   1:  PR[GP1:91,2] = PR[GP1:90,2] + -38.074;
   1:L PR[91] 10mm/sec CNT100;
   1:  PR[GP1:91,1] = PR[GP1:90,1] + -20.726;
   1:  PR[GP1:91,2] = PR[GP1:90,2] + -40.892;
   1:L PR[91] 10mm/sec CNT100;
   1:  PR[GP1:91,1] = PR[GP1:90,1] + -15.398;
   1:  PR[GP1:91,2] = PR[GP1:90,2] + -40.986;
   1:L PR[91] 10mm/sec CNT100;
   1:  PR[GP1:91,1] = PR[GP1:90,1] + -5.344;
   1:  PR[GP1:91,2] = PR[GP1:90,2] + -40.628;
   1:L PR[91] 10mm/sec CNT100;
   1:  PR[GP1:91,1] = PR[GP1:90,1] + -1.074;
   1:  PR[GP1:91,2] = PR[GP1:90,2] + -39.306;
   1:L PR[91] 10mm/sec CNT100;
   1:  PR[GP1:91,1] = PR[GP1:90,1] + 1.895;
   1:  PR[GP1:91,2] = PR[GP1:90,2] + -39.305;
   1:L PR[91] 10mm/sec CNT100;
   1:  PR[GP1:91,1] = PR[GP1:90,1] + 6.165;
   1:  PR[GP1:91,2] = PR[GP1:90,2] + -40.627;
   1:L PR[91] 10mm/sec CNT100;
   1:  PR[GP1:91,1] = PR[GP1:90,1] + 16.219;
   1:  PR[GP1:91,2] = PR[GP1:90,2] + -40.986;
   1:L PR[91] 10mm/sec CNT100;
   1:  PR[GP1:91,1] = PR[GP1:90,1] + 21.547;
   1:  PR[GP1:91,2] = PR[GP1:90,2] + -40.892;
   1:L PR[91] 10mm/sec CNT100;
   1:  PR[GP1:91,1] = PR[GP1:90,1] + 30.135;
   1:  PR[GP1:91,2] = PR[GP1:90,2] + -38.074;
   1:L PR[91] 10mm/sec CNT100;
   1:  PR[GP1:91,1] = PR[GP1:90,1] + 35.902;
   1:  PR[GP1:91,2] = PR[GP1:90,2] + -35.950;
   1:L PR[91] 10mm/sec CNT100;
   1:  PR[GP1:91,1] = PR[GP1:90,1] + 42.200;
   1:  PR[GP1:91,2] = PR[GP1:90,2] + -30.964;
   1:L PR[91] 10mm/sec CNT100;
   1:  PR[GP1:91,1] = PR[GP1:90,1] + 47.482;
   1:  PR[GP1:91,2] = PR[GP1:90,2] + -26.602;
   1:L PR[91] 10mm/sec CNT100;
   1:  PR[GP1:91,1] = PR[GP1:90,1] + 51.199;
   1:  PR[GP1:91,2] = PR[GP1:90,2] + -20.456;
   1:L PR[91] 10mm/sec CNT100;
   1:  PR[GP1:91,1] = PR[GP1:90,1] + 54.958;
   1:  PR[GP1:91,2] = PR[GP1:90,2] + -14.112;
   1:L PR[91] 10mm/sec CNT100;
   1:  PR[GP1:91,1] = PR[GP1:90,1] + 56.363;
   1:  PR[GP1:91,2] = PR[GP1:90,2] + -6.354;
   1:L PR[91] 10mm/sec CNT100;
   1:  PR[GP1:91,1] = PR[GP1:90,1] + 57.385;
   1:  PR[GP1:91,2] = PR[GP1:90,2] + -0.011;
   1:L PR[91] 10mm/sec CNT100;
   1:  PR[GP1:91,1] = PR[GP1:90,1] + 56.882;
   1:  PR[GP1:91,2] = PR[GP1:90,2] + 2.758;
   1:L PR[91] 10mm/sec CNT100;
   1:  PR[GP1:91,1] = PR[GP1:90,1] + 56.158;
   1:  PR[GP1:91,2] = PR[GP1:90,2] + 7.602;
   1:L PR[91] 10mm/sec CNT100;
   1:  PR[GP1:91,1] = PR[GP1:90,1] + 54.959;
   1:  PR[GP1:91,2] = PR[GP1:90,2] + 14.100;
   1:L PR[91] 10mm/sec CNT100;
   1:  PR[GP1:91,1] = PR[GP1:90,1] + 51.202;
   1:  PR[GP1:91,2] = PR[GP1:90,2] + 20.445;
   1:L PR[91] 10mm/sec CNT100;
   1:  PR[GP1:91,1] = PR[GP1:90,1] + 47.484;
   1:  PR[GP1:91,2] = PR[GP1:90,2] + 26.591;
   1:L PR[91] 10mm/sec CNT100;
   1:  PR[GP1:91,1] = PR[GP1:90,1] + 42.205;
   1:  PR[GP1:91,2] = PR[GP1:90,2] + 30.953;
   1:L PR[91] 10mm/sec CNT100;
   1:  PR[GP1:91,1] = PR[GP1:90,1] + 35.906;
   1:  PR[GP1:91,2] = PR[GP1:90,2] + 35.939;
   1:L PR[91] 10mm/sec CNT100;
   1:  PR[GP1:91,1] = PR[GP1:90,1] + 30.141;
   1:  PR[GP1:91,2] = PR[GP1:90,2] + 38.065;
   1:L PR[91] 10mm/sec CNT100;
   1:  PR[GP1:91,1] = PR[GP1:90,1] + 21.552;
   1:  PR[GP1:91,2] = PR[GP1:90,2] + 40.882;
   1:L PR[91] 10mm/sec CNT100;
   1:  PR[GP1:91,1] = PR[GP1:90,1] + 16.224;
   1:  PR[GP1:91,2] = PR[GP1:90,2] + 40.978;
   1:L PR[91] 10mm/sec CNT100;
   1:  PR[GP1:91,1] = PR[GP1:90,1] + 6.166;
   1:  PR[GP1:91,2] = PR[GP1:90,2] + 40.618;
   1:L PR[91] 10mm/sec CNT100;
   1:  PR[GP1:91,1] = PR[GP1:90,1] + 1.894;
   1:  PR[GP1:91,2] = PR[GP1:90,2] + 39.305;
   1:L PR[91] 10mm/sec CNT100;
   1:  PR[GP1:91,1] = PR[GP1:90,1] + -1.017;
   1:  PR[GP1:91,2] = PR[GP1:90,2] + 39.683;
   1:  PR[GP1:91,3] = PR[GP1:90,3] + 91.770;
   1:L PR[91] 10mm/sec CNT100;
   1:  PR[GP1:91,1] = PR[GP1:90,1] + -4.695;
   1:  PR[GP1:91,2] = PR[GP1:90,2] + 40.812;
   1:L PR[91] 10mm/sec CNT100;
   1:  PR[GP1:91,1] = PR[GP1:90,1] + -15.487;
   1:  PR[GP1:91,2] = PR[GP1:90,2] + 41.199;
   1:L PR[91] 10mm/sec CNT100;
   1:  PR[GP1:91,1] = PR[GP1:90,1] + -20.161;
   1:  PR[GP1:91,2] = PR[GP1:90,2] + 41.113;
   1:L PR[91] 10mm/sec CNT100;
   1:  PR[GP1:91,1] = PR[GP1:90,1] + -29.470;
   1:  PR[GP1:91,2] = PR[GP1:90,2] + 38.060;
   1:L PR[91] 10mm/sec CNT100;
   1:  PR[GP1:91,1] = PR[GP1:90,1] + -34.602;
   1:  PR[GP1:91,2] = PR[GP1:90,2] + 36.166;
   1:L PR[91] 10mm/sec CNT100;
   1:  PR[GP1:91,1] = PR[GP1:90,1] + -41.515;
   1:  PR[GP1:91,2] = PR[GP1:90,2] + 30.696;
   1:L PR[91] 10mm/sec CNT100;
   1:  PR[GP1:91,1] = PR[GP1:90,1] + -46.261;
   1:  PR[GP1:91,2] = PR[GP1:90,2] + 26.779;
   1:L PR[91] 10mm/sec CNT100;
   1:  PR[GP1:91,1] = PR[GP1:90,1] + -50.396;
   1:  PR[GP1:91,2] = PR[GP1:90,2] + 19.939;
   1:L PR[91] 10mm/sec CNT100;
   1:  PR[GP1:91,1] = PR[GP1:90,1] + -53.792;
   1:  PR[GP1:91,2] = PR[GP1:90,2] + 14.192;
   1:L PR[91] 10mm/sec CNT100;
   1:  PR[GP1:91,1] = PR[GP1:90,1] + -55.062;
   1:  PR[GP1:91,2] = PR[GP1:90,2] + 7.190;
   1:L PR[91] 10mm/sec CNT100;
   1:  PR[GP1:91,1] = PR[GP1:90,1] + -56.220;
   1:  PR[GP1:91,2] = PR[GP1:90,2] + 0.002;
   1:L PR[91] 10mm/sec CNT100;
   1:  PR[GP1:91,1] = PR[GP1:90,1] + -55.955;
   1:  PR[GP1:91,2] = PR[GP1:90,2] + -1.459;
   1:L PR[91] 10mm/sec CNT100;
   1:  PR[GP1:91,1] = PR[GP1:90,1] + -55.141;
   1:  PR[GP1:91,2] = PR[GP1:90,2] + -6.893;
   1:L PR[91] 10mm/sec CNT100;
   1:  PR[GP1:91,1] = PR[GP1:90,1] + -53.792;
   1:  PR[GP1:91,2] = PR[GP1:90,2] + -14.202;
   1:L PR[91] 10mm/sec CNT100;
   1:  PR[GP1:91,1] = PR[GP1:90,1] + -50.394;
   1:  PR[GP1:91,2] = PR[GP1:90,2] + -19.950;
   1:L PR[91] 10mm/sec CNT100;
   1:  PR[GP1:91,1] = PR[GP1:90,1] + -46.259;
   1:  PR[GP1:91,2] = PR[GP1:90,2] + -26.790;
   1:L PR[91] 10mm/sec CNT100;
   1:  PR[GP1:91,1] = PR[GP1:90,1] + -41.511;
   1:  PR[GP1:91,2] = PR[GP1:90,2] + -30.707;
   1:L PR[91] 10mm/sec CNT100;
   1:  PR[GP1:91,1] = PR[GP1:90,1] + -34.598;
   1:  PR[GP1:91,2] = PR[GP1:90,2] + -36.177;
   1:L PR[91] 10mm/sec CNT100;
   1:  PR[GP1:91,1] = PR[GP1:90,1] + -29.465;
   1:  PR[GP1:91,2] = PR[GP1:90,2] + -38.069;
   1:L PR[91] 10mm/sec CNT100;
   1:  PR[GP1:91,1] = PR[GP1:90,1] + -20.157;
   1:  PR[GP1:91,2] = PR[GP1:90,2] + -41.123;
   1:L PR[91] 10mm/sec CNT100;
   1:  PR[GP1:91,1] = PR[GP1:90,1] + -15.482;
   1:  PR[GP1:91,2] = PR[GP1:90,2] + -41.206;
   1:L PR[91] 10mm/sec CNT100;
   1:  PR[GP1:91,1] = PR[GP1:90,1] + -4.696;
   1:  PR[GP1:91,2] = PR[GP1:90,2] + -40.821;
   1:L PR[91] 10mm/sec CNT100;
   1:  PR[GP1:91,1] = PR[GP1:90,1] + -1.019;
   1:  PR[GP1:91,2] = PR[GP1:90,2] + -39.684;
   1:L PR[91] 10mm/sec CNT100;
   1:  PR[GP1:91,1] = PR[GP1:90,1] + 1.841;
   1:L PR[91] 10mm/sec CNT100;
   1:  PR[GP1:91,1] = PR[GP1:90,1] + 5.518;
   1:  PR[GP1:91,2] = PR[GP1:90,2] + -40.821;
   1:L PR[91] 10mm/sec CNT100;
   1:  PR[GP1:91,1] = PR[GP1:90,1] + 16.304;
   1:  PR[GP1:91,2] = PR[GP1:90,2] + -41.205;
   1:L PR[91] 10mm/sec CNT100;
   1:  PR[GP1:91,1] = PR[GP1:90,1] + 20.979;
   1:  PR[GP1:91,2] = PR[GP1:90,2] + -41.123;
   1:L PR[91] 10mm/sec CNT100;
   1:  PR[GP1:91,1] = PR[GP1:90,1] + 30.286;
   1:  PR[GP1:91,2] = PR[GP1:90,2] + -38.069;
   1:L PR[91] 10mm/sec CNT100;
   1:  PR[GP1:91,1] = PR[GP1:90,1] + 35.419;
   1:  PR[GP1:91,2] = PR[GP1:90,2] + -36.178;
   1:L PR[91] 10mm/sec CNT100;
   1:  PR[GP1:91,1] = PR[GP1:90,1] + 42.331;
   1:  PR[GP1:91,2] = PR[GP1:90,2] + -30.706;
   1:L PR[91] 10mm/sec CNT100;
   1:  PR[GP1:91,1] = PR[GP1:90,1] + 47.079;
   1:  PR[GP1:91,2] = PR[GP1:90,2] + -26.786;
   1:L PR[91] 10mm/sec CNT100;
   1:  PR[GP1:91,1] = PR[GP1:90,1] + 51.215;
   1:  PR[GP1:91,2] = PR[GP1:90,2] + -19.949;
   1:L PR[91] 10mm/sec CNT100;
   1:  PR[GP1:91,1] = PR[GP1:90,1] + 54.612;
   1:  PR[GP1:91,2] = PR[GP1:90,2] + -14.214;
   1:L PR[91] 10mm/sec CNT100;
   1:  PR[GP1:91,1] = PR[GP1:90,1] + 55.883;
   1:  PR[GP1:91,2] = PR[GP1:90,2] + -7.201;
   1:L PR[91] 10mm/sec CNT100;
   1:  PR[GP1:91,1] = PR[GP1:90,1] + 57.041;
   1:  PR[GP1:91,2] = PR[GP1:90,2] + -0.011;
   1:L PR[91] 10mm/sec CNT100;
   1:  PR[GP1:91,1] = PR[GP1:90,1] + 56.775;
   1:  PR[GP1:91,2] = PR[GP1:90,2] + 1.452;
   1:L PR[91] 10mm/sec CNT100;
   1:  PR[GP1:91,1] = PR[GP1:90,1] + 55.962;
   1:  PR[GP1:91,2] = PR[GP1:90,2] + 6.892;
   1:L PR[91] 10mm/sec CNT100;
   1:  PR[GP1:91,1] = PR[GP1:90,1] + 54.614;
   1:  PR[GP1:91,2] = PR[GP1:90,2] + 14.203;
   1:L PR[91] 10mm/sec CNT100;
   1:  PR[GP1:91,1] = PR[GP1:90,1] + 51.217;
   1:  PR[GP1:91,2] = PR[GP1:90,2] + 19.938;
   1:L PR[91] 10mm/sec CNT100;
   1:  PR[GP1:91,1] = PR[GP1:90,1] + 47.081;
   1:  PR[GP1:91,2] = PR[GP1:90,2] + 26.774;
   1:L PR[91] 10mm/sec CNT100;
   1:  PR[GP1:91,1] = PR[GP1:90,1] + 42.335;
   1:  PR[GP1:91,2] = PR[GP1:90,2] + 30.696;
   1:L PR[91] 10mm/sec CNT100;
   1:  PR[GP1:91,1] = PR[GP1:90,1] + 35.423;
   1:  PR[GP1:91,2] = PR[GP1:90,2] + 36.168;
   1:L PR[91] 10mm/sec CNT100;
   1:  PR[GP1:91,1] = PR[GP1:90,1] + 30.290;
   1:  PR[GP1:91,2] = PR[GP1:90,2] + 38.060;
   1:L PR[91] 10mm/sec CNT100;
   1:  PR[GP1:91,1] = PR[GP1:90,1] + 20.982;
   1:  PR[GP1:91,2] = PR[GP1:90,2] + 41.113;
   1:L PR[91] 10mm/sec CNT100;
   1:  PR[GP1:91,1] = PR[GP1:90,1] + 16.308;
   1:  PR[GP1:91,2] = PR[GP1:90,2] + 41.198;
   1:L PR[91] 10mm/sec CNT100;
   1:  PR[GP1:91,1] = PR[GP1:90,1] + 5.517;
   1:  PR[GP1:91,2] = PR[GP1:90,2] + 40.811;
   1:L PR[91] 10mm/sec CNT100;
   1:  PR[GP1:91,1] = PR[GP1:90,1] + 1.839;
   1:  PR[GP1:91,2] = PR[GP1:90,2] + 39.683;
   1:L PR[91] 10mm/sec CNT100;
   1:  PR[GP1:91,1] = PR[GP1:90,1] + -0.962;
   1:  PR[GP1:91,2] = PR[GP1:90,2] + 40.061;
   1:  PR[GP1:91,3] = PR[GP1:90,3] + 93.100;
   1:L PR[91] 10mm/sec CNT100;
   1:  PR[GP1:91,1] = PR[GP1:90,1] + -4.046;
   1:  PR[GP1:91,2] = PR[GP1:90,2] + 41.005;
   1:L PR[91] 10mm/sec CNT100;
   1:  PR[GP1:91,1] = PR[GP1:90,1] + -15.570;
   1:  PR[GP1:91,2] = PR[GP1:90,2] + 41.418;
   1:L PR[91] 10mm/sec CNT100;
   1:  PR[GP1:91,1] = PR[GP1:90,1] + -19.591;
   1:  PR[GP1:91,2] = PR[GP1:90,2] + 41.345;
   1:L PR[91] 10mm/sec CNT100;
   1:  PR[GP1:91,1] = PR[GP1:90,1] + -29.619;
   1:  PR[GP1:91,2] = PR[GP1:90,2] + 38.056;
   1:L PR[91] 10mm/sec CNT100;
   1:  PR[GP1:91,1] = PR[GP1:90,1] + -34.119;
   1:  PR[GP1:91,2] = PR[GP1:90,2] + 36.395;
   1:L PR[91] 10mm/sec CNT100;
   1:  PR[GP1:91,1] = PR[GP1:90,1] + -41.646;
   1:  PR[GP1:91,2] = PR[GP1:90,2] + 30.439;
   1:L PR[91] 10mm/sec CNT100;
   1:  PR[GP1:91,1] = PR[GP1:90,1] + -45.858;
   1:  PR[GP1:91,2] = PR[GP1:90,2] + 26.962;
   1:L PR[91] 10mm/sec CNT100;
   1:  PR[GP1:91,1] = PR[GP1:90,1] + -50.412;
   1:  PR[GP1:91,2] = PR[GP1:90,2] + 19.431;
   1:L PR[91] 10mm/sec CNT100;
   1:  PR[GP1:91,1] = PR[GP1:90,1] + -53.447;
   1:  PR[GP1:91,2] = PR[GP1:90,2] + 14.295;
   1:L PR[91] 10mm/sec CNT100;
   1:  PR[GP1:91,1] = PR[GP1:90,1] + -54.582;
   1:  PR[GP1:91,2] = PR[GP1:90,2] + 8.036;
   1:L PR[91] 10mm/sec CNT100;
   1:  PR[GP1:91,1] = PR[GP1:90,1] + -55.878;
   1:  PR[GP1:91,2] = PR[GP1:90,2] + -0.007;
   1:L PR[91] 10mm/sec CNT100;
   1:  PR[GP1:91,1] = PR[GP1:90,1] + -54.945;
   1:  PR[GP1:91,2] = PR[GP1:90,2] + -6.182;
   1:L PR[91] 10mm/sec CNT100;
   1:  PR[GP1:91,1] = PR[GP1:90,1] + -53.447;
   1:  PR[GP1:91,2] = PR[GP1:90,2] + -14.304;
   1:L PR[91] 10mm/sec CNT100;
   1:  PR[GP1:91,1] = PR[GP1:90,1] + -50.409;
   1:  PR[GP1:91,2] = PR[GP1:90,2] + -19.442;
   1:L PR[91] 10mm/sec CNT100;
   1:  PR[GP1:91,1] = PR[GP1:90,1] + -45.856;
   1:  PR[GP1:91,2] = PR[GP1:90,2] + -26.973;
   1:L PR[91] 10mm/sec CNT100;
   1:  PR[GP1:91,1] = PR[GP1:90,1] + -41.642;
   1:  PR[GP1:91,2] = PR[GP1:90,2] + -30.450;
   1:L PR[91] 10mm/sec CNT100;
   1:  PR[GP1:91,1] = PR[GP1:90,1] + -34.116;
   1:  PR[GP1:91,2] = PR[GP1:90,2] + -36.406;
   1:L PR[91] 10mm/sec CNT100;
   1:  PR[GP1:91,1] = PR[GP1:90,1] + -29.615;
   1:  PR[GP1:91,2] = PR[GP1:90,2] + -38.065;
   1:L PR[91] 10mm/sec CNT100;
   1:  PR[GP1:91,1] = PR[GP1:90,1] + -19.588;
   1:  PR[GP1:91,2] = PR[GP1:90,2] + -41.354;
   1:L PR[91] 10mm/sec CNT100;
   1:  PR[GP1:91,1] = PR[GP1:90,1] + -15.567;
   1:  PR[GP1:91,2] = PR[GP1:90,2] + -41.425;
   1:L PR[91] 10mm/sec CNT100;
   1:  PR[GP1:91,1] = PR[GP1:90,1] + -4.049;
   1:  PR[GP1:91,2] = PR[GP1:90,2] + -41.015;
   1:L PR[91] 10mm/sec CNT100;
   1:  PR[GP1:91,1] = PR[GP1:90,1] + -0.964;
   1:  PR[GP1:91,2] = PR[GP1:90,2] + -40.063;
   1:L PR[91] 10mm/sec CNT100;
   1:  PR[GP1:91,1] = PR[GP1:90,1] + 1.786;
   1:L PR[91] 10mm/sec CNT100;
   1:  PR[GP1:91,1] = PR[GP1:90,1] + 4.871;
   1:  PR[GP1:91,2] = PR[GP1:90,2] + -41.015;
   1:L PR[91] 10mm/sec CNT100;
   1:  PR[GP1:91,1] = PR[GP1:90,1] + 16.388;
   1:  PR[GP1:91,2] = PR[GP1:90,2] + -41.425;
   1:L PR[91] 10mm/sec CNT100;
   1:  PR[GP1:91,1] = PR[GP1:90,1] + 20.410;
   1:  PR[GP1:91,2] = PR[GP1:90,2] + -41.354;
   1:L PR[91] 10mm/sec CNT100;
   1:  PR[GP1:91,1] = PR[GP1:90,1] + 30.436;
   1:  PR[GP1:91,2] = PR[GP1:90,2] + -38.065;
   1:L PR[91] 10mm/sec CNT100;
   1:  PR[GP1:91,1] = PR[GP1:90,1] + 34.937;
   1:  PR[GP1:91,2] = PR[GP1:90,2] + -36.407;
   1:L PR[91] 10mm/sec CNT100;
   1:  PR[GP1:91,1] = PR[GP1:90,1] + 42.463;
   1:  PR[GP1:91,2] = PR[GP1:90,2] + -30.449;
   1:L PR[91] 10mm/sec CNT100;
   1:  PR[GP1:91,1] = PR[GP1:90,1] + 46.677;
   1:  PR[GP1:91,2] = PR[GP1:90,2] + -26.969;
   1:L PR[91] 10mm/sec CNT100;
   1:  PR[GP1:91,1] = PR[GP1:90,1] + 51.230;
   1:  PR[GP1:91,2] = PR[GP1:90,2] + -19.442;
   1:L PR[91] 10mm/sec CNT100;
   1:  PR[GP1:91,1] = PR[GP1:90,1] + 54.267;
   1:  PR[GP1:91,2] = PR[GP1:90,2] + -14.316;
   1:L PR[91] 10mm/sec CNT100;
   1:  PR[GP1:91,1] = PR[GP1:90,1] + 55.403;
   1:  PR[GP1:91,2] = PR[GP1:90,2] + -8.047;
   1:L PR[91] 10mm/sec CNT100;
   1:  PR[GP1:91,1] = PR[GP1:90,1] + 56.699;
   1:  PR[GP1:91,2] = PR[GP1:90,2] + -0.001;
   1:L PR[91] 10mm/sec CNT100;
   1:  PR[GP1:91,1] = PR[GP1:90,1] + 55.767;
   1:  PR[GP1:91,2] = PR[GP1:90,2] + 6.180;
   1:L PR[91] 10mm/sec CNT100;
   1:  PR[GP1:91,1] = PR[GP1:90,1] + 54.268;
   1:  PR[GP1:91,2] = PR[GP1:90,2] + 14.305;
   1:L PR[91] 10mm/sec CNT100;
   1:  PR[GP1:91,1] = PR[GP1:90,1] + 51.232;
   1:  PR[GP1:91,2] = PR[GP1:90,2] + 19.431;
   1:L PR[91] 10mm/sec CNT100;
   1:  PR[GP1:91,1] = PR[GP1:90,1] + 46.679;
   1:  PR[GP1:91,2] = PR[GP1:90,2] + 26.958;
   1:L PR[91] 10mm/sec CNT100;
   1:  PR[GP1:91,1] = PR[GP1:90,1] + 42.466;
   1:  PR[GP1:91,2] = PR[GP1:90,2] + 30.439;
   1:L PR[91] 10mm/sec CNT100;
   1:  PR[GP1:91,1] = PR[GP1:90,1] + 34.940;
   1:  PR[GP1:91,2] = PR[GP1:90,2] + 36.396;
   1:L PR[91] 10mm/sec CNT100;
   1:  PR[GP1:91,1] = PR[GP1:90,1] + 30.440;
   1:  PR[GP1:91,2] = PR[GP1:90,2] + 38.056;
   1:L PR[91] 10mm/sec CNT100;
   1:  PR[GP1:91,1] = PR[GP1:90,1] + 20.413;
   1:  PR[GP1:91,2] = PR[GP1:90,2] + 41.345;
   1:L PR[91] 10mm/sec CNT100;
   1:  PR[GP1:91,1] = PR[GP1:90,1] + 16.391;
   1:  PR[GP1:91,2] = PR[GP1:90,2] + 41.418;
   1:L PR[91] 10mm/sec CNT100;
   1:  PR[GP1:91,1] = PR[GP1:90,1] + 4.868;
   1:  PR[GP1:91,2] = PR[GP1:90,2] + 41.005;
   1:L PR[91] 10mm/sec CNT100;
   1:  PR[GP1:91,1] = PR[GP1:90,1] + 1.784;
   1:  PR[GP1:91,2] = PR[GP1:90,2] + 40.061;
   1:L PR[91] 10mm/sec CNT100;
   1:  PR[GP1:91,1] = PR[GP1:90,1] + -0.907;
   1:  PR[GP1:91,2] = PR[GP1:90,2] + 40.438;
   1:  PR[GP1:91,3] = PR[GP1:90,3] + 94.430;
   1:L PR[91] 10mm/sec CNT100;
   1:  PR[GP1:91,1] = PR[GP1:90,1] + -3.397;
   1:  PR[GP1:91,2] = PR[GP1:90,2] + 41.198;
   1:L PR[91] 10mm/sec CNT100;
   1:  PR[GP1:91,1] = PR[GP1:90,1] + -15.653;
   1:  PR[GP1:91,2] = PR[GP1:90,2] + 41.638;
   1:L PR[91] 10mm/sec CNT100;
   1:  PR[GP1:91,1] = PR[GP1:90,1] + -19.021;
   1:  PR[GP1:91,2] = PR[GP1:90,2] + 41.576;
   1:L PR[91] 10mm/sec CNT100;
   1:  PR[GP1:91,1] = PR[GP1:90,1] + -29.768;
   1:  PR[GP1:91,2] = PR[GP1:90,2] + 38.052;
   1:L PR[91] 10mm/sec CNT100;
   1:  PR[GP1:91,1] = PR[GP1:90,1] + -33.636;
   1:  PR[GP1:91,2] = PR[GP1:90,2] + 36.624;
   1:L PR[91] 10mm/sec CNT100;
   1:  PR[GP1:91,1] = PR[GP1:90,1] + -41.776;
   1:  PR[GP1:91,2] = PR[GP1:90,2] + 30.183;
   1:L PR[91] 10mm/sec CNT100;
   1:  PR[GP1:91,1] = PR[GP1:90,1] + -45.455;
   1:  PR[GP1:91,2] = PR[GP1:90,2] + 27.146;
   1:L PR[91] 10mm/sec CNT100;
   1:  PR[GP1:91,1] = PR[GP1:90,1] + -50.427;
   1:  PR[GP1:91,2] = PR[GP1:90,2] + 18.924;
   1:L PR[91] 10mm/sec CNT100;
   1:  PR[GP1:91,1] = PR[GP1:90,1] + -53.101;
   1:  PR[GP1:91,2] = PR[GP1:90,2] + 14.398;
   1:L PR[91] 10mm/sec CNT100;
   1:  PR[GP1:91,1] = PR[GP1:90,1] + -54.101;
   1:  PR[GP1:91,2] = PR[GP1:90,2] + 8.883;
   1:L PR[91] 10mm/sec CNT100;
   1:  PR[GP1:91,1] = PR[GP1:90,1] + -55.310;
   1:  PR[GP1:91,2] = PR[GP1:90,2] + 1.381;
   1:L PR[91] 10mm/sec CNT100;
   1:  PR[GP1:91,1] = PR[GP1:90,1] + -55.567;
   1:  PR[GP1:91,2] = PR[GP1:90,2] + -0.015;
   1:L PR[91] 10mm/sec CNT100;
   1:  PR[GP1:91,1] = PR[GP1:90,1] + -54.750;
   1:  PR[GP1:91,2] = PR[GP1:90,2] + -5.473;
   1:L PR[91] 10mm/sec CNT100;
   1:  PR[GP1:91,1] = PR[GP1:90,1] + -53.101;
   1:  PR[GP1:91,2] = PR[GP1:90,2] + -14.407;
   1:L PR[91] 10mm/sec CNT100;
   1:  PR[GP1:91,1] = PR[GP1:90,1] + -50.425;
   1:  PR[GP1:91,2] = PR[GP1:90,2] + -18.935;
   1:L PR[91] 10mm/sec CNT100;
   1:  PR[GP1:91,1] = PR[GP1:90,1] + -45.454;
   1:  PR[GP1:91,2] = PR[GP1:90,2] + -27.156;
   1:L PR[91] 10mm/sec CNT100;
   1:  PR[GP1:91,1] = PR[GP1:90,1] + -41.773;
   1:  PR[GP1:91,2] = PR[GP1:90,2] + -30.193;
   1:L PR[91] 10mm/sec CNT100;
   1:  PR[GP1:91,1] = PR[GP1:90,1] + -33.634;
   1:  PR[GP1:91,2] = PR[GP1:90,2] + -36.634;
   1:L PR[91] 10mm/sec CNT100;
   1:  PR[GP1:91,1] = PR[GP1:90,1] + -29.765;
   1:  PR[GP1:91,2] = PR[GP1:90,2] + -38.060;
   1:L PR[91] 10mm/sec CNT100;
   1:  PR[GP1:91,1] = PR[GP1:90,1] + -19.020;
   1:  PR[GP1:91,2] = PR[GP1:90,2] + -41.585;
   1:L PR[91] 10mm/sec CNT100;
   1:  PR[GP1:91,1] = PR[GP1:90,1] + -15.651;
   1:  PR[GP1:91,2] = PR[GP1:90,2] + -41.645;
   1:L PR[91] 10mm/sec CNT100;
   1:  PR[GP1:91,1] = PR[GP1:90,1] + -3.401;
   1:  PR[GP1:91,2] = PR[GP1:90,2] + -41.208;
   1:L PR[91] 10mm/sec CNT100;
   1:  PR[GP1:91,1] = PR[GP1:90,1] + -0.908;
   1:  PR[GP1:91,2] = PR[GP1:90,2] + -40.442;
   1:L PR[91] 10mm/sec CNT100;
   1:  PR[GP1:91,1] = PR[GP1:90,1] + 1.731;
   1:  PR[GP1:91,2] = PR[GP1:90,2] + -40.441;
   1:L PR[91] 10mm/sec CNT100;
   1:  PR[GP1:91,1] = PR[GP1:90,1] + 4.224;
   1:  PR[GP1:91,2] = PR[GP1:90,2] + -41.208;
   1:L PR[91] 10mm/sec CNT100;
   1:  PR[GP1:91,1] = PR[GP1:90,1] + 16.473;
   1:  PR[GP1:91,2] = PR[GP1:90,2] + -41.645;
   1:L PR[91] 10mm/sec CNT100;
   1:  PR[GP1:91,1] = PR[GP1:90,1] + 19.842;
   1:  PR[GP1:91,2] = PR[GP1:90,2] + -41.585;
   1:L PR[91] 10mm/sec CNT100;
   1:  PR[GP1:91,1] = PR[GP1:90,1] + 30.586;
   1:  PR[GP1:91,2] = PR[GP1:90,2] + -38.060;
   1:L PR[91] 10mm/sec CNT100;
   1:  PR[GP1:91,1] = PR[GP1:90,1] + 34.455;
   1:  PR[GP1:91,2] = PR[GP1:90,2] + -36.635;
   1:L PR[91] 10mm/sec CNT100;
   1:  PR[GP1:91,1] = PR[GP1:90,1] + 42.594;
   1:  PR[GP1:91,2] = PR[GP1:90,2] + -30.192;
   1:L PR[91] 10mm/sec CNT100;
   1:  PR[GP1:91,1] = PR[GP1:90,1] + 46.275;
   1:  PR[GP1:91,2] = PR[GP1:90,2] + -27.152;
   1:L PR[91] 10mm/sec CNT100;
   1:  PR[GP1:91,1] = PR[GP1:90,1] + 51.246;
   1:  PR[GP1:91,2] = PR[GP1:90,2] + -18.934;
   1:L PR[91] 10mm/sec CNT100;
   1:  PR[GP1:91,1] = PR[GP1:90,1] + 53.922;
   1:  PR[GP1:91,2] = PR[GP1:90,2] + -14.418;
   1:L PR[91] 10mm/sec CNT100;
   1:  PR[GP1:91,1] = PR[GP1:90,1] + 54.922;
   1:  PR[GP1:91,2] = PR[GP1:90,2] + -8.894;
   1:L PR[91] 10mm/sec CNT100;
   1:  PR[GP1:91,1] = PR[GP1:90,1] + 56.131;
   1:  PR[GP1:91,2] = PR[GP1:90,2] + -1.390;
   1:L PR[91] 10mm/sec CNT100;
   1:  PR[GP1:91,1] = PR[GP1:90,1] + 56.388;
   1:  PR[GP1:91,2] = PR[GP1:90,2] + 0.006;
   1:L PR[91] 10mm/sec CNT100;
   1:  PR[GP1:91,1] = PR[GP1:90,1] + 55.571;
   1:  PR[GP1:91,2] = PR[GP1:90,2] + 5.470;
   1:L PR[91] 10mm/sec CNT100;
   1:  PR[GP1:91,1] = PR[GP1:90,1] + 53.922;
   1:  PR[GP1:91,2] = PR[GP1:90,2] + 14.407;
   1:L PR[91] 10mm/sec CNT100;
   1:  PR[GP1:91,1] = PR[GP1:90,1] + 51.248;
   1:  PR[GP1:91,2] = PR[GP1:90,2] + 18.924;
   1:L PR[91] 10mm/sec CNT100;
   1:  PR[GP1:91,1] = PR[GP1:90,1] + 46.276;
   1:  PR[GP1:91,2] = PR[GP1:90,2] + 27.142;
   1:L PR[91] 10mm/sec CNT100;
   1:  PR[GP1:91,1] = PR[GP1:90,1] + 42.596;
   1:  PR[GP1:91,2] = PR[GP1:90,2] + 30.182;
   1:L PR[91] 10mm/sec CNT100;
   1:  PR[GP1:91,1] = PR[GP1:90,1] + 34.457;
   1:  PR[GP1:91,2] = PR[GP1:90,2] + 36.625;
   1:L PR[91] 10mm/sec CNT100;
   1:  PR[GP1:91,1] = PR[GP1:90,1] + 30.589;
   1:  PR[GP1:91,2] = PR[GP1:90,2] + 38.051;
   1:L PR[91] 10mm/sec CNT100;
   1:  PR[GP1:91,1] = PR[GP1:90,1] + 19.843;
   1:  PR[GP1:91,2] = PR[GP1:90,2] + 41.576;
   1:L PR[91] 10mm/sec CNT100;
   1:  PR[GP1:91,1] = PR[GP1:90,1] + 16.475;
   1:  PR[GP1:91,2] = PR[GP1:90,2] + 41.637;
   1:L PR[91] 10mm/sec CNT100;
   1:  PR[GP1:91,1] = PR[GP1:90,1] + 4.220;
   1:  PR[GP1:91,2] = PR[GP1:90,2] + 41.198;
   1:L PR[91] 10mm/sec CNT100;
   1:  PR[GP1:91,1] = PR[GP1:90,1] + 1.729;
   1:  PR[GP1:91,2] = PR[GP1:90,2] + 40.438;
   1:L PR[91] 10mm/sec CNT100;
   1:  PR[GP1:91,1] = PR[GP1:90,1] + -0.851;
   1:  PR[GP1:91,2] = PR[GP1:90,2] + 40.816;
   1:  PR[GP1:91,3] = PR[GP1:90,3] + 95.760;
   1:L PR[91] 10mm/sec CNT100;
   1:  PR[GP1:91,1] = PR[GP1:90,1] + -2.748;
   1:  PR[GP1:91,2] = PR[GP1:90,2] + 41.391;
   1:L PR[91] 10mm/sec CNT100;
   1:  PR[GP1:91,1] = PR[GP1:90,1] + -15.736;
   1:  PR[GP1:91,2] = PR[GP1:90,2] + 41.857;
   1:L PR[91] 10mm/sec CNT100;
   1:  PR[GP1:91,1] = PR[GP1:90,1] + -18.451;
   1:  PR[GP1:91,2] = PR[GP1:90,2] + 41.807;
   1:L PR[91] 10mm/sec CNT100;
   1:  PR[GP1:91,1] = PR[GP1:90,1] + -29.917;
   1:  PR[GP1:91,2] = PR[GP1:90,2] + 38.047;
   1:L PR[91] 10mm/sec CNT100;
   1:  PR[GP1:91,1] = PR[GP1:90,1] + -33.153;
   1:  PR[GP1:91,2] = PR[GP1:90,2] + 36.853;
   1:L PR[91] 10mm/sec CNT100;
   1:  PR[GP1:91,1] = PR[GP1:90,1] + -41.907;
   1:  PR[GP1:91,2] = PR[GP1:90,2] + 29.926;
   1:L PR[91] 10mm/sec CNT100;
   1:  PR[GP1:91,1] = PR[GP1:90,1] + -45.053;
   1:  PR[GP1:91,2] = PR[GP1:90,2] + 27.329;
   1:L PR[91] 10mm/sec CNT100;
   1:  PR[GP1:91,1] = PR[GP1:90,1] + -50.442;
   1:  PR[GP1:91,2] = PR[GP1:90,2] + 18.416;
   1:L PR[91] 10mm/sec CNT100;
   1:  PR[GP1:91,1] = PR[GP1:90,1] + -52.756;
   1:  PR[GP1:91,2] = PR[GP1:90,2] + 14.501;
   1:L PR[91] 10mm/sec CNT100;
   1:  PR[GP1:91,1] = PR[GP1:90,1] + -53.621;
   1:  PR[GP1:91,2] = PR[GP1:90,2] + 9.729;
   1:L PR[91] 10mm/sec CNT100;
   1:  PR[GP1:91,1] = PR[GP1:90,1] + -54.670;
   1:  PR[GP1:91,2] = PR[GP1:90,2] + 3.218;
   1:L PR[91] 10mm/sec CNT100;
   1:  PR[GP1:91,1] = PR[GP1:90,1] + -55.265;
   1:  PR[GP1:91,2] = PR[GP1:90,2] + -0.015;
   1:L PR[91] 10mm/sec CNT100;
   1:  PR[GP1:91,1] = PR[GP1:90,1] + -54.554;
   1:  PR[GP1:91,2] = PR[GP1:90,2] + -4.763;
   1:L PR[91] 10mm/sec CNT100;
   1:  PR[GP1:91,1] = PR[GP1:90,1] + -52.756;
   1:  PR[GP1:91,2] = PR[GP1:90,2] + -14.510;
   1:L PR[91] 10mm/sec CNT100;
   1:  PR[GP1:91,1] = PR[GP1:90,1] + -50.440;
   1:  PR[GP1:91,2] = PR[GP1:90,2] + -18.427;
   1:L PR[91] 10mm/sec CNT100;
   1:  PR[GP1:91,1] = PR[GP1:90,1] + -45.052;
   1:  PR[GP1:91,2] = PR[GP1:90,2] + -27.339;
   1:L PR[91] 10mm/sec CNT100;
   1:  PR[GP1:91,1] = PR[GP1:90,1] + -41.904;
   1:  PR[GP1:91,2] = PR[GP1:90,2] + -29.936;
   1:L PR[91] 10mm/sec CNT100;
   1:  PR[GP1:91,1] = PR[GP1:90,1] + -33.151;
   1:  PR[GP1:91,2] = PR[GP1:90,2] + -36.863;
   1:L PR[91] 10mm/sec CNT100;
   1:  PR[GP1:91,1] = PR[GP1:90,1] + -29.915;
   1:  PR[GP1:91,2] = PR[GP1:90,2] + -38.056;
   1:L PR[91] 10mm/sec CNT100;
   1:  PR[GP1:91,1] = PR[GP1:90,1] + -18.451;
   1:  PR[GP1:91,2] = PR[GP1:90,2] + -41.817;
   1:L PR[91] 10mm/sec CNT100;
   1:  PR[GP1:91,1] = PR[GP1:90,1] + -15.736;
   1:  PR[GP1:91,2] = PR[GP1:90,2] + -41.865;
   1:L PR[91] 10mm/sec CNT100;
   1:  PR[GP1:91,1] = PR[GP1:90,1] + -2.753;
   1:  PR[GP1:91,2] = PR[GP1:90,2] + -41.402;
   1:L PR[91] 10mm/sec CNT100;
   1:  PR[GP1:91,1] = PR[GP1:90,1] + -0.853;
   1:  PR[GP1:91,2] = PR[GP1:90,2] + -40.820;
   1:L PR[91] 10mm/sec CNT100;
   1:  PR[GP1:91,1] = PR[GP1:90,1] + 1.676;
   1:L PR[91] 10mm/sec CNT100;
   1:  PR[GP1:91,1] = PR[GP1:90,1] + 3.576;
   1:  PR[GP1:91,2] = PR[GP1:90,2] + -41.402;
   1:L PR[91] 10mm/sec CNT100;
   1:  PR[GP1:91,1] = PR[GP1:90,1] + 16.558;
   1:  PR[GP1:91,2] = PR[GP1:90,2] + -41.864;
   1:L PR[91] 10mm/sec CNT100;
   1:  PR[GP1:91,1] = PR[GP1:90,1] + 19.273;
   1:  PR[GP1:91,2] = PR[GP1:90,2] + -41.817;
   1:L PR[91] 10mm/sec CNT100;
   1:  PR[GP1:91,1] = PR[GP1:90,1] + 30.737;
   1:  PR[GP1:91,2] = PR[GP1:90,2] + -38.056;
   1:L PR[91] 10mm/sec CNT100;
   1:  PR[GP1:91,1] = PR[GP1:90,1] + 33.973;
   1:  PR[GP1:91,2] = PR[GP1:90,2] + -36.863;
   1:L PR[91] 10mm/sec CNT100;
   1:  PR[GP1:91,1] = PR[GP1:90,1] + 42.725;
   1:  PR[GP1:91,2] = PR[GP1:90,2] + -29.935;
   1:L PR[91] 10mm/sec CNT100;
   1:  PR[GP1:91,1] = PR[GP1:90,1] + 45.873;
   1:  PR[GP1:91,2] = PR[GP1:90,2] + -27.335;
   1:L PR[91] 10mm/sec CNT100;
   1:  PR[GP1:91,1] = PR[GP1:90,1] + 51.261;
   1:  PR[GP1:91,2] = PR[GP1:90,2] + -18.427;
   1:L PR[91] 10mm/sec CNT100;
   1:  PR[GP1:91,1] = PR[GP1:90,1] + 53.576;
   1:  PR[GP1:91,2] = PR[GP1:90,2] + -14.520;
   1:L PR[91] 10mm/sec CNT100;
   1:  PR[GP1:91,1] = PR[GP1:90,1] + 54.442;
   1:  PR[GP1:91,2] = PR[GP1:90,2] + -9.740;
   1:L PR[91] 10mm/sec CNT100;
   1:  PR[GP1:91,1] = PR[GP1:90,1] + 55.491;
   1:  PR[GP1:91,2] = PR[GP1:90,2] + -3.228;
   1:L PR[91] 10mm/sec CNT100;
   1:  PR[GP1:91,1] = PR[GP1:90,1] + 56.086;
   1:  PR[GP1:91,2] = PR[GP1:90,2] + 0.006;
   1:L PR[91] 10mm/sec CNT100;
   1:  PR[GP1:91,1] = PR[GP1:90,1] + 55.375;
   1:  PR[GP1:91,2] = PR[GP1:90,2] + 4.760;
   1:L PR[91] 10mm/sec CNT100;
   1:  PR[GP1:91,1] = PR[GP1:90,1] + 53.577;
   1:  PR[GP1:91,2] = PR[GP1:90,2] + 14.509;
   1:L PR[91] 10mm/sec CNT100;
   1:  PR[GP1:91,1] = PR[GP1:90,1] + 51.263;
   1:  PR[GP1:91,2] = PR[GP1:90,2] + 18.417;
   1:L PR[91] 10mm/sec CNT100;
   1:  PR[GP1:91,1] = PR[GP1:90,1] + 45.874;
   1:  PR[GP1:91,2] = PR[GP1:90,2] + 27.325;
   1:L PR[91] 10mm/sec CNT100;
   1:  PR[GP1:91,1] = PR[GP1:90,1] + 42.727;
   1:  PR[GP1:91,2] = PR[GP1:90,2] + 29.925;
   1:L PR[91] 10mm/sec CNT100;
   1:  PR[GP1:91,1] = PR[GP1:90,1] + 33.974;
   1:  PR[GP1:91,2] = PR[GP1:90,2] + 36.854;
   1:L PR[91] 10mm/sec CNT100;
   1:  PR[GP1:91,1] = PR[GP1:90,1] + 30.739;
   1:  PR[GP1:91,2] = PR[GP1:90,2] + 38.047;
   1:L PR[91] 10mm/sec CNT100;
   1:  PR[GP1:91,1] = PR[GP1:90,1] + 19.273;
   1:  PR[GP1:91,2] = PR[GP1:90,2] + 41.807;
   1:L PR[91] 10mm/sec CNT100;
   1:  PR[GP1:91,1] = PR[GP1:90,1] + 16.559;
   1:  PR[GP1:91,2] = PR[GP1:90,2] + 41.857;
   1:L PR[91] 10mm/sec CNT100;
   1:  PR[GP1:91,1] = PR[GP1:90,1] + 3.571;
   1:  PR[GP1:91,2] = PR[GP1:90,2] + 41.391;
   1:L PR[91] 10mm/sec CNT100;
   1:  PR[GP1:91,1] = PR[GP1:90,1] + 1.674;
   1:  PR[GP1:91,2] = PR[GP1:90,2] + 40.816;
   1:L PR[91] 10mm/sec CNT100;
   1:  PR[GP1:91,1] = PR[GP1:90,1] + -0.795;
   1:  PR[GP1:91,2] = PR[GP1:90,2] + 41.194;
   1:  PR[GP1:91,3] = PR[GP1:90,3] + 97.090;
   1:L PR[91] 10mm/sec CNT100;
   1:  PR[GP1:91,1] = PR[GP1:90,1] + -2.098;
   1:  PR[GP1:91,2] = PR[GP1:90,2] + 41.584;
   1:L PR[91] 10mm/sec CNT100;
   1:  PR[GP1:91,1] = PR[GP1:90,1] + -15.820;
   1:  PR[GP1:91,2] = PR[GP1:90,2] + 42.077;
   1:L PR[91] 10mm/sec CNT100;
   1:  PR[GP1:91,1] = PR[GP1:90,1] + -17.881;
   1:  PR[GP1:91,2] = PR[GP1:90,2] + 42.039;
   1:L PR[91] 10mm/sec CNT100;
   1:  PR[GP1:91,1] = PR[GP1:90,1] + -30.066;
   1:  PR[GP1:91,2] = PR[GP1:90,2] + 38.043;
   1:L PR[91] 10mm/sec CNT100;
   1:  PR[GP1:91,1] = PR[GP1:90,1] + -32.669;
   1:  PR[GP1:91,2] = PR[GP1:90,2] + 37.082;
   1:L PR[91] 10mm/sec CNT100;
   1:  PR[GP1:91,1] = PR[GP1:90,1] + -42.037;
   1:  PR[GP1:91,2] = PR[GP1:90,2] + 29.669;
   1:L PR[91] 10mm/sec CNT100;
   1:  PR[GP1:91,1] = PR[GP1:90,1] + -44.650;
   1:  PR[GP1:91,2] = PR[GP1:90,2] + 27.513;
   1:L PR[91] 10mm/sec CNT100;
   1:  PR[GP1:91,1] = PR[GP1:90,1] + -50.457;
   1:  PR[GP1:91,2] = PR[GP1:90,2] + 17.909;
   1:L PR[91] 10mm/sec CNT100;
   1:  PR[GP1:91,1] = PR[GP1:90,1] + -52.410;
   1:  PR[GP1:91,2] = PR[GP1:90,2] + 14.604;
   1:L PR[91] 10mm/sec CNT100;
   1:  PR[GP1:91,1] = PR[GP1:90,1] + -53.141;
   1:  PR[GP1:91,2] = PR[GP1:90,2] + 10.575;
   1:L PR[91] 10mm/sec CNT100;
   1:  PR[GP1:91,1] = PR[GP1:90,1] + -54.030;
   1:  PR[GP1:91,2] = PR[GP1:90,2] + 5.055;
   1:L PR[91] 10mm/sec CNT100;
   1:  PR[GP1:91,1] = PR[GP1:90,1] + -54.963;
   1:  PR[GP1:91,2] = PR[GP1:90,2] + -0.015;
   1:L PR[91] 10mm/sec CNT100;
   1:  PR[GP1:91,1] = PR[GP1:90,1] + -54.359;
   1:  PR[GP1:91,2] = PR[GP1:90,2] + -4.053;
   1:L PR[91] 10mm/sec CNT100;
   1:  PR[GP1:91,1] = PR[GP1:90,1] + -52.410;
   1:  PR[GP1:91,2] = PR[GP1:90,2] + -14.612;
   1:L PR[91] 10mm/sec CNT100;
   1:  PR[GP1:91,1] = PR[GP1:90,1] + -50.456;
   1:  PR[GP1:91,2] = PR[GP1:90,2] + -17.919;
   1:L PR[91] 10mm/sec CNT100;
   1:  PR[GP1:91,1] = PR[GP1:90,1] + -44.650;
   1:  PR[GP1:91,2] = PR[GP1:90,2] + -27.522;
   1:L PR[91] 10mm/sec CNT100;
   1:  PR[GP1:91,1] = PR[GP1:90,1] + -42.035;
   1:  PR[GP1:91,2] = PR[GP1:90,2] + -29.679;
   1:L PR[91] 10mm/sec CNT100;
   1:  PR[GP1:91,1] = PR[GP1:90,1] + -32.669;
   1:  PR[GP1:91,2] = PR[GP1:90,2] + -37.091;
   1:L PR[91] 10mm/sec CNT100;
   1:  PR[GP1:91,1] = PR[GP1:90,1] + -30.066;
   1:  PR[GP1:91,2] = PR[GP1:90,2] + -38.051;
   1:L PR[91] 10mm/sec CNT100;
   1:  PR[GP1:91,1] = PR[GP1:90,1] + -17.882;
   1:  PR[GP1:91,2] = PR[GP1:90,2] + -42.048;
   1:L PR[91] 10mm/sec CNT100;
   1:  PR[GP1:91,1] = PR[GP1:90,1] + -15.820;
   1:  PR[GP1:91,2] = PR[GP1:90,2] + -42.084;
   1:L PR[91] 10mm/sec CNT100;
   1:  PR[GP1:91,1] = PR[GP1:90,1] + -2.105;
   1:  PR[GP1:91,2] = PR[GP1:90,2] + -41.595;
   1:L PR[91] 10mm/sec CNT100;
   1:  PR[GP1:91,1] = PR[GP1:90,1] + -0.797;
   1:  PR[GP1:91,2] = PR[GP1:90,2] + -41.199;
   1:L PR[91] 10mm/sec CNT100;
   1:  PR[GP1:91,1] = PR[GP1:90,1] + 1.620;
   1:L PR[91] 10mm/sec CNT100;
   1:  PR[GP1:91,1] = PR[GP1:90,1] + 2.928;
   1:  PR[GP1:91,2] = PR[GP1:90,2] + -41.595;
   1:L PR[91] 10mm/sec CNT100;
   1:  PR[GP1:91,1] = PR[GP1:90,1] + 16.642;
   1:  PR[GP1:91,2] = PR[GP1:90,2] + -42.084;
   1:L PR[91] 10mm/sec CNT100;
   1:  PR[GP1:91,1] = PR[GP1:90,1] + 18.705;
   1:  PR[GP1:91,2] = PR[GP1:90,2] + -42.048;
   1:L PR[91] 10mm/sec CNT100;
   1:  PR[GP1:91,1] = PR[GP1:90,1] + 30.887;
   1:  PR[GP1:91,2] = PR[GP1:90,2] + -38.051;
   1:L PR[91] 10mm/sec CNT100;
   1:  PR[GP1:91,1] = PR[GP1:90,1] + 33.491;
   1:  PR[GP1:91,2] = PR[GP1:90,2] + -37.092;
   1:L PR[91] 10mm/sec CNT100;
   1:  PR[GP1:91,1] = PR[GP1:90,1] + 42.856;
   1:  PR[GP1:91,2] = PR[GP1:90,2] + -29.677;
   1:L PR[91] 10mm/sec CNT100;
   1:  PR[GP1:91,1] = PR[GP1:90,1] + 45.471;
   1:  PR[GP1:91,2] = PR[GP1:90,2] + -27.518;
   1:L PR[91] 10mm/sec CNT100;
   1:  PR[GP1:91,1] = PR[GP1:90,1] + 51.277;
   1:  PR[GP1:91,2] = PR[GP1:90,2] + -17.920;
   1:L PR[91] 10mm/sec CNT100;
   1:  PR[GP1:91,1] = PR[GP1:90,1] + 53.231;
   1:  PR[GP1:91,2] = PR[GP1:90,2] + -14.622;
   1:L PR[91] 10mm/sec CNT100;
   1:  PR[GP1:91,1] = PR[GP1:90,1] + 53.962;
   1:  PR[GP1:91,2] = PR[GP1:90,2] + -10.586;
   1:L PR[91] 10mm/sec CNT100;
   1:  PR[GP1:91,1] = PR[GP1:90,1] + 54.851;
   1:  PR[GP1:91,2] = PR[GP1:90,2] + -5.065;
   1:L PR[91] 10mm/sec CNT100;
   1:  PR[GP1:91,1] = PR[GP1:90,1] + 55.784;
   1:  PR[GP1:91,2] = PR[GP1:90,2] + 0.006;
   1:L PR[91] 10mm/sec CNT100;
   1:  PR[GP1:91,1] = PR[GP1:90,1] + 55.180;
   1:  PR[GP1:91,2] = PR[GP1:90,2] + 4.049;
   1:L PR[91] 10mm/sec CNT100;
   1:  PR[GP1:91,1] = PR[GP1:90,1] + 53.231;
   1:  PR[GP1:91,2] = PR[GP1:90,2] + 14.612;
   1:L PR[91] 10mm/sec CNT100;
   1:  PR[GP1:91,1] = PR[GP1:90,1] + 51.278;
   1:  PR[GP1:91,2] = PR[GP1:90,2] + 17.910;
   1:L PR[91] 10mm/sec CNT100;
   1:  PR[GP1:91,1] = PR[GP1:90,1] + 45.471;
   1:  PR[GP1:91,2] = PR[GP1:90,2] + 27.509;
   1:L PR[91] 10mm/sec CNT100;
   1:  PR[GP1:91,1] = PR[GP1:90,1] + 42.858;
   1:  PR[GP1:91,2] = PR[GP1:90,2] + 29.668;
   1:L PR[91] 10mm/sec CNT100;
   1:  PR[GP1:91,1] = PR[GP1:90,1] + 33.491;
   1:  PR[GP1:91,2] = PR[GP1:90,2] + 37.083;
   1:L PR[91] 10mm/sec CNT100;
   1:  PR[GP1:91,1] = PR[GP1:90,1] + 30.888;
   1:  PR[GP1:91,2] = PR[GP1:90,2] + 38.043;
   1:L PR[91] 10mm/sec CNT100;
   1:  PR[GP1:91,1] = PR[GP1:90,1] + 18.704;
   1:  PR[GP1:91,2] = PR[GP1:90,2] + 42.039;
   1:L PR[91] 10mm/sec CNT100;
   1:  PR[GP1:91,1] = PR[GP1:90,1] + 16.642;
   1:  PR[GP1:91,2] = PR[GP1:90,2] + 42.076;
   1:L PR[91] 10mm/sec CNT100;
   1:  PR[GP1:91,1] = PR[GP1:90,1] + 2.921;
   1:  PR[GP1:91,2] = PR[GP1:90,2] + 41.584;
   1:L PR[91] 10mm/sec CNT100;
   1:  PR[GP1:91,1] = PR[GP1:90,1] + 1.619;
   1:  PR[GP1:91,2] = PR[GP1:90,2] + 41.194;
   1:L PR[91] 10mm/sec CNT100;
   1:  PR[GP1:91,1] = PR[GP1:90,1] + -0.738;
   1:  PR[GP1:91,2] = PR[GP1:90,2] + 41.571;
   1:  PR[GP1:91,3] = PR[GP1:90,3] + 98.420;
   1:L PR[91] 10mm/sec CNT100;
   1:  PR[GP1:91,1] = PR[GP1:90,1] + -1.447;
   1:  PR[GP1:91,2] = PR[GP1:90,2] + 41.778;
   1:L PR[91] 10mm/sec CNT100;
   1:  PR[GP1:91,1] = PR[GP1:90,1] + -15.903;
   1:  PR[GP1:91,2] = PR[GP1:90,2] + 42.296;
   1:L PR[91] 10mm/sec CNT100;
   1:  PR[GP1:91,1] = PR[GP1:90,1] + -17.311;
   1:  PR[GP1:91,2] = PR[GP1:90,2] + 42.270;
   1:L PR[91] 10mm/sec CNT100;
   1:  PR[GP1:91,1] = PR[GP1:90,1] + -30.216;
   1:  PR[GP1:91,2] = PR[GP1:90,2] + 38.038;
   1:L PR[91] 10mm/sec CNT100;
   1:  PR[GP1:91,1] = PR[GP1:90,1] + -32.186;
   1:  PR[GP1:91,2] = PR[GP1:90,2] + 37.311;
   1:L PR[91] 10mm/sec CNT100;
   1:  PR[GP1:91,1] = PR[GP1:90,1] + -42.168;
   1:  PR[GP1:91,2] = PR[GP1:90,2] + 29.413;
   1:L PR[91] 10mm/sec CNT100;
   1:  PR[GP1:91,1] = PR[GP1:90,1] + -44.247;
   1:  PR[GP1:91,2] = PR[GP1:90,2] + 27.696;
   1:L PR[91] 10mm/sec CNT100;
   1:  PR[GP1:91,1] = PR[GP1:90,1] + -50.472;
   1:  PR[GP1:91,2] = PR[GP1:90,2] + 17.401;
   1:L PR[91] 10mm/sec CNT100;
   1:  PR[GP1:91,1] = PR[GP1:90,1] + -52.064;
   1:  PR[GP1:91,2] = PR[GP1:90,2] + 14.707;
   1:L PR[91] 10mm/sec CNT100;
   1:  PR[GP1:91,1] = PR[GP1:90,1] + -52.660;
   1:  PR[GP1:91,2] = PR[GP1:90,2] + 11.421;
   1:L PR[91] 10mm/sec CNT100;
   1:  PR[GP1:91,1] = PR[GP1:90,1] + -53.390;
   1:  PR[GP1:91,2] = PR[GP1:90,2] + 6.892;
   1:L PR[91] 10mm/sec CNT100;
   1:  PR[GP1:91,1] = PR[GP1:90,1] + -54.662;
   1:  PR[GP1:91,2] = PR[GP1:90,2] + -0.015;
   1:L PR[91] 10mm/sec CNT100;
   1:  PR[GP1:91,1] = PR[GP1:90,1] + -54.163;
   1:  PR[GP1:91,2] = PR[GP1:90,2] + -3.343;
   1:L PR[91] 10mm/sec CNT100;
   1:  PR[GP1:91,1] = PR[GP1:90,1] + -52.065;
   1:  PR[GP1:91,2] = PR[GP1:90,2] + -14.715;
   1:L PR[91] 10mm/sec CNT100;
   1:  PR[GP1:91,1] = PR[GP1:90,1] + -50.471;
   1:  PR[GP1:91,2] = PR[GP1:90,2] + -17.411;
   1:L PR[91] 10mm/sec CNT100;
   1:  PR[GP1:91,1] = PR[GP1:90,1] + -44.247;
   1:  PR[GP1:91,2] = PR[GP1:90,2] + -27.705;
   1:L PR[91] 10mm/sec CNT100;
   1:  PR[GP1:91,1] = PR[GP1:90,1] + -42.166;
   1:  PR[GP1:91,2] = PR[GP1:90,2] + -29.422;
   1:L PR[91] 10mm/sec CNT100;
   1:  PR[GP1:91,1] = PR[GP1:90,1] + -32.187;
   1:  PR[GP1:91,2] = PR[GP1:90,2] + -37.320;
   1:L PR[91] 10mm/sec CNT100;
   1:  PR[GP1:91,1] = PR[GP1:90,1] + -30.216;
   1:  PR[GP1:91,2] = PR[GP1:90,2] + -38.046;
   1:L PR[91] 10mm/sec CNT100;
   1:  PR[GP1:91,1] = PR[GP1:90,1] + -17.313;
   1:  PR[GP1:91,2] = PR[GP1:90,2] + -42.279;
   1:L PR[91] 10mm/sec CNT100;
   1:  PR[GP1:91,1] = PR[GP1:90,1] + -15.904;
   1:  PR[GP1:91,2] = PR[GP1:90,2] + -42.304;
   1:L PR[91] 10mm/sec CNT100;
   1:  PR[GP1:91,1] = PR[GP1:90,1] + -1.455;
   1:  PR[GP1:91,2] = PR[GP1:90,2] + -41.789;
   1:L PR[91] 10mm/sec CNT100;
   1:  PR[GP1:91,1] = PR[GP1:90,1] + -0.739;
   1:  PR[GP1:91,2] = PR[GP1:90,2] + -41.578;
   1:L PR[91] 10mm/sec CNT100;
   1:  PR[GP1:91,1] = PR[GP1:90,1] + 1.563;
   1:L PR[91] 10mm/sec CNT100;
   1:  PR[GP1:91,1] = PR[GP1:90,1] + 2.279;
   1:  PR[GP1:91,2] = PR[GP1:90,2] + -41.789;
   1:L PR[91] 10mm/sec CNT100;
   1:  PR[GP1:91,1] = PR[GP1:90,1] + 16.727;
   1:  PR[GP1:91,2] = PR[GP1:90,2] + -42.304;
   1:L PR[91] 10mm/sec CNT100;
   1:  PR[GP1:91,1] = PR[GP1:90,1] + 18.136;
   1:  PR[GP1:91,2] = PR[GP1:90,2] + -42.279;
   1:L PR[91] 10mm/sec CNT100;
   1:  PR[GP1:91,1] = PR[GP1:90,1] + 31.037;
   1:  PR[GP1:91,2] = PR[GP1:90,2] + -38.046;
   1:L PR[91] 10mm/sec CNT100;
   1:  PR[GP1:91,1] = PR[GP1:90,1] + 33.009;
   1:  PR[GP1:91,2] = PR[GP1:90,2] + -37.320;
   1:L PR[91] 10mm/sec CNT100;
   1:  PR[GP1:91,1] = PR[GP1:90,1] + 42.988;
   1:  PR[GP1:91,2] = PR[GP1:90,2] + -29.420;
   1:L PR[91] 10mm/sec CNT100;
   1:  PR[GP1:91,1] = PR[GP1:90,1] + 45.069;
   1:  PR[GP1:91,2] = PR[GP1:90,2] + -27.702;
   1:L PR[91] 10mm/sec CNT100;
   1:  PR[GP1:91,1] = PR[GP1:90,1] + 51.292;
   1:  PR[GP1:91,2] = PR[GP1:90,2] + -17.413;
   1:L PR[91] 10mm/sec CNT100;
   1:  PR[GP1:91,1] = PR[GP1:90,1] + 52.885;
   1:  PR[GP1:91,2] = PR[GP1:90,2] + -14.724;
   1:L PR[91] 10mm/sec CNT100;
   1:  PR[GP1:91,1] = PR[GP1:90,1] + 53.481;
   1:  PR[GP1:91,2] = PR[GP1:90,2] + -11.433;
   1:L PR[91] 10mm/sec CNT100;
   1:  PR[GP1:91,1] = PR[GP1:90,1] + 54.211;
   1:  PR[GP1:91,2] = PR[GP1:90,2] + -6.903;
   1:L PR[91] 10mm/sec CNT100;
   1:  PR[GP1:91,1] = PR[GP1:90,1] + 55.482;
   1:  PR[GP1:91,2] = PR[GP1:90,2] + 0.006;
   1:L PR[91] 10mm/sec CNT100;
   1:  PR[GP1:91,1] = PR[GP1:90,1] + 54.984;
   1:  PR[GP1:91,2] = PR[GP1:90,2] + 3.338;
   1:L PR[91] 10mm/sec CNT100;
   1:  PR[GP1:91,1] = PR[GP1:90,1] + 52.886;
   1:  PR[GP1:91,2] = PR[GP1:90,2] + 14.714;
   1:L PR[91] 10mm/sec CNT100;
   1:  PR[GP1:91,1] = PR[GP1:90,1] + 51.293;
   1:  PR[GP1:91,2] = PR[GP1:90,2] + 17.403;
   1:L PR[91] 10mm/sec CNT100;
   1:  PR[GP1:91,1] = PR[GP1:90,1] + 45.069;
   1:  PR[GP1:91,2] = PR[GP1:90,2] + 27.693;
   1:L PR[91] 10mm/sec CNT100;
   1:  PR[GP1:91,1] = PR[GP1:90,1] + 42.988;
   1:  PR[GP1:91,2] = PR[GP1:90,2] + 29.412;
   1:L PR[91] 10mm/sec CNT100;
   1:  PR[GP1:91,1] = PR[GP1:90,1] + 33.008;
   1:  PR[GP1:91,2] = PR[GP1:90,2] + 37.311;
   1:L PR[91] 10mm/sec CNT100;
   1:  PR[GP1:91,1] = PR[GP1:90,1] + 31.038;
   1:  PR[GP1:91,2] = PR[GP1:90,2] + 38.038;
   1:L PR[91] 10mm/sec CNT100;
   1:  PR[GP1:91,1] = PR[GP1:90,1] + 18.134;
   1:  PR[GP1:91,2] = PR[GP1:90,2] + 42.270;
   1:L PR[91] 10mm/sec CNT100;
   1:  PR[GP1:91,1] = PR[GP1:90,1] + 16.726;
   1:  PR[GP1:91,2] = PR[GP1:90,2] + 42.296;
   1:L PR[91] 10mm/sec CNT100;
   1:  PR[GP1:91,1] = PR[GP1:90,1] + 2.270;
   1:  PR[GP1:91,2] = PR[GP1:90,2] + 41.778;
   1:L PR[91] 10mm/sec CNT100;
   1:  PR[GP1:91,1] = PR[GP1:90,1] + 1.561;
   1:  PR[GP1:91,2] = PR[GP1:90,2] + 41.571;
   1:L PR[91] 10mm/sec CNT100;
   1:  PR[GP1:91,1] = PR[GP1:90,1] + -0.679;
   1:  PR[GP1:91,2] = PR[GP1:90,2] + 41.940;
   1:  PR[GP1:91,3] = PR[GP1:90,3] + 99.750;
   1:L PR[91] 10mm/sec CNT100;
   1:  PR[GP1:91,1] = PR[GP1:90,1] + -0.792;
   1:  PR[GP1:91,2] = PR[GP1:90,2] + 41.971;
   1:L PR[91] 10mm/sec CNT100;
   1:  PR[GP1:91,1] = PR[GP1:90,1] + -15.986;
   1:  PR[GP1:91,2] = PR[GP1:90,2] + 42.516;
   1:L PR[91] 10mm/sec CNT100;
   1:  PR[GP1:91,1] = PR[GP1:90,1] + -16.742;
   1:  PR[GP1:91,2] = PR[GP1:90,2] + 42.502;
   1:L PR[91] 10mm/sec CNT100;
   1:  PR[GP1:91,1] = PR[GP1:90,1] + -30.365;
   1:  PR[GP1:91,2] = PR[GP1:90,2] + 38.034;
   1:L PR[91] 10mm/sec CNT100;
   1:  PR[GP1:91,1] = PR[GP1:90,1] + -31.703;
   1:  PR[GP1:91,2] = PR[GP1:90,2] + 37.540;
   1:L PR[91] 10mm/sec CNT100;
   1:  PR[GP1:91,1] = PR[GP1:90,1] + -42.298;
   1:  PR[GP1:91,2] = PR[GP1:90,2] + 29.156;
   1:L PR[91] 10mm/sec CNT100;
   1:  PR[GP1:91,1] = PR[GP1:90,1] + -43.845;
   1:  PR[GP1:91,2] = PR[GP1:90,2] + 27.880;
   1:L PR[91] 10mm/sec CNT100;
   1:  PR[GP1:91,1] = PR[GP1:90,1] + -50.487;
   1:  PR[GP1:91,2] = PR[GP1:90,2] + 16.894;
   1:L PR[91] 10mm/sec CNT100;
   1:  PR[GP1:91,1] = PR[GP1:90,1] + -51.719;
   1:  PR[GP1:91,2] = PR[GP1:90,2] + 14.810;
   1:L PR[91] 10mm/sec CNT100;
   1:  PR[GP1:91,1] = PR[GP1:90,1] + -52.180;
   1:  PR[GP1:91,2] = PR[GP1:90,2] + 12.267;
   1:L PR[91] 10mm/sec CNT100;
   1:  PR[GP1:91,1] = PR[GP1:90,1] + -52.750;
   1:  PR[GP1:91,2] = PR[GP1:90,2] + 8.729;
   1:L PR[91] 10mm/sec CNT100;
   1:  PR[GP1:91,1] = PR[GP1:90,1] + -54.360;
   1:  PR[GP1:91,2] = PR[GP1:90,2] + -0.015;
   1:L PR[91] 10mm/sec CNT100;
   1:  PR[GP1:91,1] = PR[GP1:90,1] + -53.968;
   1:  PR[GP1:91,2] = PR[GP1:90,2] + -2.633;
   1:L PR[91] 10mm/sec CNT100;
   1:  PR[GP1:91,1] = PR[GP1:90,1] + -51.719;
   1:  PR[GP1:91,2] = PR[GP1:90,2] + -14.818;
   1:L PR[91] 10mm/sec CNT100;
   1:  PR[GP1:91,1] = PR[GP1:90,1] + -50.486;
   1:  PR[GP1:91,2] = PR[GP1:90,2] + -16.903;
   1:L PR[91] 10mm/sec CNT100;
   1:  PR[GP1:91,1] = PR[GP1:90,1] + -43.845;
   1:  PR[GP1:91,2] = PR[GP1:90,2] + -27.888;
   1:L PR[91] 10mm/sec CNT100;
   1:  PR[GP1:91,1] = PR[GP1:90,1] + -42.297;
   1:  PR[GP1:91,2] = PR[GP1:90,2] + -29.165;
   1:L PR[91] 10mm/sec CNT100;
   1:  PR[GP1:91,1] = PR[GP1:90,1] + -31.705;
   1:  PR[GP1:91,2] = PR[GP1:90,2] + -37.548;
   1:L PR[91] 10mm/sec CNT100;
   1:  PR[GP1:91,1] = PR[GP1:90,1] + -30.366;
   1:  PR[GP1:91,2] = PR[GP1:90,2] + -38.042;
   1:L PR[91] 10mm/sec CNT100;
   1:  PR[GP1:91,1] = PR[GP1:90,1] + -16.744;
   1:  PR[GP1:91,2] = PR[GP1:90,2] + -42.510;
   1:L PR[91] 10mm/sec CNT100;
   1:  PR[GP1:91,1] = PR[GP1:90,1] + -15.989;
   1:  PR[GP1:91,2] = PR[GP1:90,2] + -42.524;
   1:L PR[91] 10mm/sec CNT100;
   1:  PR[GP1:91,1] = PR[GP1:90,1] + -0.801;
   1:  PR[GP1:91,2] = PR[GP1:90,2] + -41.982;
   1:L PR[91] 10mm/sec CNT100;
   1:  PR[GP1:91,1] = PR[GP1:90,1] + -0.679;
   1:  PR[GP1:91,2] = PR[GP1:90,2] + -41.949;
   1:L PR[91] 10mm/sec CNT100;
   1:  PR[GP1:91,1] = PR[GP1:90,1] + 1.502;
   1:L PR[91] 10mm/sec CNT100;
   1:  PR[GP1:91,1] = PR[GP1:90,1] + 1.625;
   1:  PR[GP1:91,2] = PR[GP1:90,2] + -41.982;
   1:L PR[91] 10mm/sec CNT100;
   1:  PR[GP1:91,1] = PR[GP1:90,1] + 16.812;
   1:  PR[GP1:91,2] = PR[GP1:90,2] + -42.523;
   1:L PR[91] 10mm/sec CNT100;
   1:  PR[GP1:91,1] = PR[GP1:90,1] + 17.568;
   1:  PR[GP1:91,2] = PR[GP1:90,2] + -42.510;
   1:L PR[91] 10mm/sec CNT100;
   1:  PR[GP1:91,1] = PR[GP1:90,1] + 31.188;
   1:  PR[GP1:91,2] = PR[GP1:90,2] + -38.042;
   1:L PR[91] 10mm/sec CNT100;
   1:  PR[GP1:91,1] = PR[GP1:90,1] + 32.527;
   1:  PR[GP1:91,2] = PR[GP1:90,2] + -37.548;
   1:L PR[91] 10mm/sec CNT100;
   1:  PR[GP1:91,1] = PR[GP1:90,1] + 43.118;
   1:  PR[GP1:91,2] = PR[GP1:90,2] + -29.163;
   1:L PR[91] 10mm/sec CNT100;
   1:  PR[GP1:91,1] = PR[GP1:90,1] + 44.666;
   1:  PR[GP1:91,2] = PR[GP1:90,2] + -27.885;
   1:L PR[91] 10mm/sec CNT100;
   1:  PR[GP1:91,1] = PR[GP1:90,1] + 51.307;
   1:  PR[GP1:91,2] = PR[GP1:90,2] + -16.906;
   1:L PR[91] 10mm/sec CNT100;
   1:  PR[GP1:91,1] = PR[GP1:90,1] + 52.540;
   1:  PR[GP1:91,2] = PR[GP1:90,2] + -14.826;
   1:L PR[91] 10mm/sec CNT100;
   1:  PR[GP1:91,1] = PR[GP1:90,1] + 53.001;
   1:  PR[GP1:91,2] = PR[GP1:90,2] + -12.279;
   1:L PR[91] 10mm/sec CNT100;
   1:  PR[GP1:91,1] = PR[GP1:90,1] + 53.571;
   1:  PR[GP1:91,2] = PR[GP1:90,2] + -8.740;
   1:L PR[91] 10mm/sec CNT100;
   1:  PR[GP1:91,1] = PR[GP1:90,1] + 55.180;
   1:  PR[GP1:91,2] = PR[GP1:90,2] + 0.006;
   1:L PR[91] 10mm/sec CNT100;
   1:  PR[GP1:91,1] = PR[GP1:90,1] + 54.788;
   1:  PR[GP1:91,2] = PR[GP1:90,2] + 2.628;
   1:L PR[91] 10mm/sec CNT100;
   1:  PR[GP1:91,1] = PR[GP1:90,1] + 52.540;
   1:  PR[GP1:91,2] = PR[GP1:90,2] + 14.816;
   1:L PR[91] 10mm/sec CNT100;
   1:  PR[GP1:91,1] = PR[GP1:90,1] + 51.308;
   1:  PR[GP1:91,2] = PR[GP1:90,2] + 16.896;
   1:L PR[91] 10mm/sec CNT100;
   1:  PR[GP1:91,1] = PR[GP1:90,1] + 44.666;
   1:  PR[GP1:91,2] = PR[GP1:90,2] + 27.876;
   1:L PR[91] 10mm/sec CNT100;
   1:  PR[GP1:91,1] = PR[GP1:90,1] + 43.119;
   1:  PR[GP1:91,2] = PR[GP1:90,2] + 29.155;
   1:L PR[91] 10mm/sec CNT100;
   1:  PR[GP1:91,1] = PR[GP1:90,1] + 32.526;
   1:  PR[GP1:91,2] = PR[GP1:90,2] + 37.540;
   1:L PR[91] 10mm/sec CNT100;
   1:  PR[GP1:91,1] = PR[GP1:90,1] + 31.187;
   1:  PR[GP1:91,2] = PR[GP1:90,2] + 38.034;
   1:L PR[91] 10mm/sec CNT100;
   1:  PR[GP1:91,1] = PR[GP1:90,1] + 17.565;
   1:  PR[GP1:91,2] = PR[GP1:90,2] + 42.502;
   1:L PR[91] 10mm/sec CNT100;
   1:  PR[GP1:91,1] = PR[GP1:90,1] + 16.809;
   1:  PR[GP1:91,2] = PR[GP1:90,2] + 42.515;
   1:L PR[91] 10mm/sec CNT100;
   1:  PR[GP1:91,1] = PR[GP1:90,1] + 1.616;
   1:  PR[GP1:91,2] = PR[GP1:90,2] + 41.971;
   1:L PR[91] 10mm/sec CNT100;
   1:  PR[GP1:91,1] = PR[GP1:90,1] + 1.502;
   1:  PR[GP1:91,2] = PR[GP1:90,2] + 41.940;
   1:L PR[91] 10mm/sec CNT100;
   1:  PR[GP1:91,1] = PR[GP1:90,1] + -0.557;
   1:  PR[GP1:91,2] = PR[GP1:90,2] + 42.289;
   1:  PR[GP1:91,3] = PR[GP1:90,3] + 101.080;
   1:L PR[91] 10mm/sec CNT100;
   1:  PR[GP1:91,1] = PR[GP1:90,1] + -11.793;
   1:  PR[GP1:91,2] = PR[GP1:90,2] + 42.582;
   1:L PR[91] 10mm/sec CNT100;
   1:  PR[GP1:91,1] = PR[GP1:90,1] + -16.069;
   1:  PR[GP1:91,2] = PR[GP1:90,2] + 42.735;
   1:L PR[91] 10mm/sec CNT100;
   1:  PR[GP1:91,1] = PR[GP1:90,1] + -16.172;
   1:  PR[GP1:91,2] = PR[GP1:90,2] + 42.733;
   1:L PR[91] 10mm/sec CNT100;
   1:  PR[GP1:91,1] = PR[GP1:90,1] + -30.514;
   1:  PR[GP1:91,2] = PR[GP1:90,2] + 38.030;
   1:L PR[91] 10mm/sec CNT100;
   1:  PR[GP1:91,1] = PR[GP1:90,1] + -31.220;
   1:  PR[GP1:91,2] = PR[GP1:90,2] + 37.769;
   1:L PR[91] 10mm/sec CNT100;
   1:  PR[GP1:91,1] = PR[GP1:90,1] + -42.429;
   1:  PR[GP1:91,2] = PR[GP1:90,2] + 28.900;
   1:L PR[91] 10mm/sec CNT100;
   1:  PR[GP1:91,1] = PR[GP1:90,1] + -43.442;
   1:  PR[GP1:91,2] = PR[GP1:90,2] + 28.063;
   1:L PR[91] 10mm/sec CNT100;
   1:  PR[GP1:91,1] = PR[GP1:90,1] + -50.503;
   1:  PR[GP1:91,2] = PR[GP1:90,2] + 16.386;
   1:L PR[91] 10mm/sec CNT100;
   1:  PR[GP1:91,1] = PR[GP1:90,1] + -51.373;
   1:  PR[GP1:91,2] = PR[GP1:90,2] + 14.913;
   1:L PR[91] 10mm/sec CNT100;
   1:  PR[GP1:91,1] = PR[GP1:90,1] + -51.699;
   1:  PR[GP1:91,2] = PR[GP1:90,2] + 13.114;
   1:L PR[91] 10mm/sec CNT100;
   1:  PR[GP1:91,1] = PR[GP1:90,1] + -52.110;
   1:  PR[GP1:91,2] = PR[GP1:90,2] + 10.566;
   1:L PR[91] 10mm/sec CNT100;
   1:  PR[GP1:91,1] = PR[GP1:90,1] + -54.058;
   1:  PR[GP1:91,2] = PR[GP1:90,2] + -0.015;
   1:L PR[91] 10mm/sec CNT100;
   1:  PR[GP1:91,1] = PR[GP1:90,1] + -53.772;
   1:  PR[GP1:91,2] = PR[GP1:90,2] + -1.924;
   1:L PR[91] 10mm/sec CNT100;
   1:  PR[GP1:91,1] = PR[GP1:90,1] + -51.374;
   1:  PR[GP1:91,2] = PR[GP1:90,2] + -14.920;
   1:L PR[91] 10mm/sec CNT100;
   1:  PR[GP1:91,1] = PR[GP1:90,1] + -50.502;
   1:  PR[GP1:91,2] = PR[GP1:90,2] + -16.395;
   1:L PR[91] 10mm/sec CNT100;
   1:  PR[GP1:91,1] = PR[GP1:90,1] + -43.443;
   1:  PR[GP1:91,2] = PR[GP1:90,2] + -28.071;
   1:L PR[91] 10mm/sec CNT100;
   1:  PR[GP1:91,1] = PR[GP1:90,1] + -42.428;
   1:  PR[GP1:91,2] = PR[GP1:90,2] + -28.908;
   1:L PR[91] 10mm/sec CNT100;
   1:  PR[GP1:91,1] = PR[GP1:90,1] + -31.222;
   1:  PR[GP1:91,2] = PR[GP1:90,2] + -37.777;
   1:L PR[91] 10mm/sec CNT100;
   1:  PR[GP1:91,1] = PR[GP1:90,1] + -30.516;
   1:  PR[GP1:91,2] = PR[GP1:90,2] + -38.037;
   1:L PR[91] 10mm/sec CNT100;
   1:  PR[GP1:91,1] = PR[GP1:90,1] + -16.176;
   1:  PR[GP1:91,2] = PR[GP1:90,2] + -42.741;
   1:L PR[91] 10mm/sec CNT100;
   1:  PR[GP1:91,1] = PR[GP1:90,1] + -16.073;
   1:  PR[GP1:91,2] = PR[GP1:90,2] + -42.743;
   1:L PR[91] 10mm/sec CNT100;
   1:  PR[GP1:91,1] = PR[GP1:90,1] + -11.729;
   1:  PR[GP1:91,2] = PR[GP1:90,2] + -42.588;
   1:L PR[91] 10mm/sec CNT100;
   1:  PR[GP1:91,1] = PR[GP1:90,1] + -0.557;
   1:  PR[GP1:91,2] = PR[GP1:90,2] + -42.297;
   1:L PR[91] 10mm/sec CNT100;
   1:  PR[GP1:91,1] = PR[GP1:90,1] + 1.380;
   1:  PR[GP1:91,2] = PR[GP1:90,2] + -42.298;
   1:L PR[91] 10mm/sec CNT100;
   1:  PR[GP1:91,1] = PR[GP1:90,1] + 12.547;
   1:  PR[GP1:91,2] = PR[GP1:90,2] + -42.588;
   1:L PR[91] 10mm/sec CNT100;
   1:  PR[GP1:91,1] = PR[GP1:90,1] + 16.896;
   1:  PR[GP1:91,2] = PR[GP1:90,2] + -42.743;
   1:L PR[91] 10mm/sec CNT100;
   1:  PR[GP1:91,1] = PR[GP1:90,1] + 16.999;
   1:  PR[GP1:91,2] = PR[GP1:90,2] + -42.741;
   1:L PR[91] 10mm/sec CNT100;
   1:  PR[GP1:91,1] = PR[GP1:90,1] + 31.338;
   1:  PR[GP1:91,2] = PR[GP1:90,2] + -38.037;
   1:L PR[91] 10mm/sec CNT100;
   1:  PR[GP1:91,1] = PR[GP1:90,1] + 32.045;
   1:  PR[GP1:91,2] = PR[GP1:90,2] + -37.777;
   1:L PR[91] 10mm/sec CNT100;
   1:  PR[GP1:91,1] = PR[GP1:90,1] + 43.250;
   1:  PR[GP1:91,2] = PR[GP1:90,2] + -28.906;
   1:L PR[91] 10mm/sec CNT100;
   1:  PR[GP1:91,1] = PR[GP1:90,1] + 44.264;
   1:  PR[GP1:91,2] = PR[GP1:90,2] + -28.068;
   1:L PR[91] 10mm/sec CNT100;
   1:  PR[GP1:91,1] = PR[GP1:90,1] + 51.323;
   1:  PR[GP1:91,2] = PR[GP1:90,2] + -16.398;
   1:L PR[91] 10mm/sec CNT100;
   1:  PR[GP1:91,1] = PR[GP1:90,1] + 52.194;
   1:  PR[GP1:91,2] = PR[GP1:90,2] + -14.928;
   1:L PR[91] 10mm/sec CNT100;
   1:  PR[GP1:91,1] = PR[GP1:90,1] + 52.521;
   1:  PR[GP1:91,2] = PR[GP1:90,2] + -13.126;
   1:L PR[91] 10mm/sec CNT100;
   1:  PR[GP1:91,1] = PR[GP1:90,1] + 52.931;
   1:  PR[GP1:91,2] = PR[GP1:90,2] + -10.578;
   1:L PR[91] 10mm/sec CNT100;
   1:  PR[GP1:91,1] = PR[GP1:90,1] + 54.878;
   1:  PR[GP1:91,2] = PR[GP1:90,2] + 0.006;
   1:L PR[91] 10mm/sec CNT100;
   1:  PR[GP1:91,1] = PR[GP1:90,1] + 54.593;
   1:  PR[GP1:91,2] = PR[GP1:90,2] + 1.917;
   1:L PR[91] 10mm/sec CNT100;
   1:  PR[GP1:91,1] = PR[GP1:90,1] + 52.195;
   1:  PR[GP1:91,2] = PR[GP1:90,2] + 14.918;
   1:L PR[91] 10mm/sec CNT100;
   1:  PR[GP1:91,1] = PR[GP1:90,1] + 51.324;
   1:  PR[GP1:91,2] = PR[GP1:90,2] + 16.389;
   1:L PR[91] 10mm/sec CNT100;
   1:  PR[GP1:91,1] = PR[GP1:90,1] + 44.264;
   1:  PR[GP1:91,2] = PR[GP1:90,2] + 28.060;
   1:L PR[91] 10mm/sec CNT100;
   1:  PR[GP1:91,1] = PR[GP1:90,1] + 43.249;
   1:  PR[GP1:91,2] = PR[GP1:90,2] + 28.898;
   1:L PR[91] 10mm/sec CNT100;
   1:  PR[GP1:91,1] = PR[GP1:90,1] + 32.043;
   1:  PR[GP1:91,2] = PR[GP1:90,2] + 37.769;
   1:L PR[91] 10mm/sec CNT100;
   1:  PR[GP1:91,1] = PR[GP1:90,1] + 31.336;
   1:  PR[GP1:91,2] = PR[GP1:90,2] + 38.029;
   1:L PR[91] 10mm/sec CNT100;
   1:  PR[GP1:91,1] = PR[GP1:90,1] + 16.995;
   1:  PR[GP1:91,2] = PR[GP1:90,2] + 42.733;
   1:L PR[91] 10mm/sec CNT100;
   1:  PR[GP1:91,1] = PR[GP1:90,1] + 16.893;
   1:  PR[GP1:91,2] = PR[GP1:90,2] + 42.735;
   1:L PR[91] 10mm/sec CNT100;
   1:  PR[GP1:91,1] = PR[GP1:90,1] + 12.611;
   1:  PR[GP1:91,2] = PR[GP1:90,2] + 42.581;
   1:L PR[91] 10mm/sec CNT100;
   1:  PR[GP1:91,1] = PR[GP1:90,1] + 1.380;
   1:  PR[GP1:91,2] = PR[GP1:90,2] + 42.289;
   1:L PR[91] 10mm/sec CNT100;
   1:  PR[GP1:91,1] = PR[GP1:90,1] + -0.508;
   1:  PR[GP1:91,2] = PR[GP1:90,2] + 42.636;
   1:  PR[GP1:91,3] = PR[GP1:90,3] + 102.410;
   1:L PR[91] 10mm/sec CNT100;
   1:  PR[GP1:91,1] = PR[GP1:90,1] + -15.512;
   1:  PR[GP1:91,2] = PR[GP1:90,2] + 43.024;
   1:L PR[91] 10mm/sec CNT100;
   1:  PR[GP1:91,1] = PR[GP1:90,1] + -15.814;
   1:  PR[GP1:91,2] = PR[GP1:90,2] + 42.987;
   1:L PR[91] 10mm/sec CNT100;
   1:  PR[GP1:91,1] = PR[GP1:90,1] + -26.448;
   1:  PR[GP1:91,2] = PR[GP1:90,2] + 39.408;
   1:L PR[91] 10mm/sec CNT100;
   1:  PR[GP1:91,1] = PR[GP1:90,1] + -30.746;
   1:  PR[GP1:91,2] = PR[GP1:90,2] + 37.991;
   1:L PR[91] 10mm/sec CNT100;
   1:  PR[GP1:91,1] = PR[GP1:90,1] + -42.559;
   1:  PR[GP1:91,2] = PR[GP1:90,2] + 28.643;
   1:L PR[91] 10mm/sec CNT100;
   1:  PR[GP1:91,1] = PR[GP1:90,1] + -43.039;
   1:  PR[GP1:91,2] = PR[GP1:90,2] + 28.247;
   1:L PR[91] 10mm/sec CNT100;
   1:  PR[GP1:91,1] = PR[GP1:90,1] + -50.517;
   1:  PR[GP1:91,2] = PR[GP1:90,2] + 15.879;
   1:L PR[91] 10mm/sec CNT100;
   1:  PR[GP1:91,1] = PR[GP1:90,1] + -51.028;
   1:  PR[GP1:91,2] = PR[GP1:90,2] + 15.015;
   1:L PR[91] 10mm/sec CNT100;
   1:  PR[GP1:91,1] = PR[GP1:90,1] + -51.219;
   1:  PR[GP1:91,2] = PR[GP1:90,2] + 13.960;
   1:L PR[91] 10mm/sec CNT100;
   1:  PR[GP1:91,1] = PR[GP1:90,1] + -51.470;
   1:  PR[GP1:91,2] = PR[GP1:90,2] + 12.403;
   1:L PR[91] 10mm/sec CNT100;
   1:  PR[GP1:91,1] = PR[GP1:90,1] + -53.756;
   1:  PR[GP1:91,2] = PR[GP1:90,2] + -0.015;
   1:L PR[91] 10mm/sec CNT100;
   1:  PR[GP1:91,1] = PR[GP1:90,1] + -53.576;
   1:  PR[GP1:91,2] = PR[GP1:90,2] + -1.214;
   1:L PR[91] 10mm/sec CNT100;
   1:  PR[GP1:91,1] = PR[GP1:90,1] + -51.028;
   1:  PR[GP1:91,2] = PR[GP1:90,2] + -15.023;
   1:L PR[91] 10mm/sec CNT100;
   1:  PR[GP1:91,1] = PR[GP1:90,1] + -50.517;
   1:  PR[GP1:91,2] = PR[GP1:90,2] + -15.888;
   1:L PR[91] 10mm/sec CNT100;
   1:  PR[GP1:91,1] = PR[GP1:90,1] + -43.041;
   1:  PR[GP1:91,2] = PR[GP1:90,2] + -28.254;
   1:L PR[91] 10mm/sec CNT100;
   1:  PR[GP1:91,1] = PR[GP1:90,1] + -42.560;
   1:  PR[GP1:91,2] = PR[GP1:90,2] + -28.651;
   1:L PR[91] 10mm/sec CNT100;
   1:  PR[GP1:91,1] = PR[GP1:90,1] + -30.748;
   1:  PR[GP1:91,2] = PR[GP1:90,2] + -37.999;
   1:L PR[91] 10mm/sec CNT100;
   1:  PR[GP1:91,1] = PR[GP1:90,1] + -26.448;
   1:  PR[GP1:91,2] = PR[GP1:90,2] + -39.416;
   1:L PR[91] 10mm/sec CNT100;
   1:  PR[GP1:91,1] = PR[GP1:90,1] + -15.818;
   1:  PR[GP1:91,2] = PR[GP1:90,2] + -42.995;
   1:L PR[91] 10mm/sec CNT100;
   1:  PR[GP1:91,1] = PR[GP1:90,1] + -15.516;
   1:  PR[GP1:91,2] = PR[GP1:90,2] + -43.032;
   1:L PR[91] 10mm/sec CNT100;
   1:  PR[GP1:91,1] = PR[GP1:90,1] + -0.508;
   1:  PR[GP1:91,2] = PR[GP1:90,2] + -42.645;
   1:L PR[91] 10mm/sec CNT100;
   1:  PR[GP1:91,1] = PR[GP1:90,1] + 1.331;
   1:L PR[91] 10mm/sec CNT100;
   1:  PR[GP1:91,1] = PR[GP1:90,1] + 16.339;
   1:  PR[GP1:91,2] = PR[GP1:90,2] + -43.032;
   1:L PR[91] 10mm/sec CNT100;
   1:  PR[GP1:91,1] = PR[GP1:90,1] + 16.641;
   1:  PR[GP1:91,2] = PR[GP1:90,2] + -42.995;
   1:L PR[91] 10mm/sec CNT100;
   1:  PR[GP1:91,1] = PR[GP1:90,1] + 27.266;
   1:  PR[GP1:91,2] = PR[GP1:90,2] + -39.418;
   1:L PR[91] 10mm/sec CNT100;
   1:  PR[GP1:91,1] = PR[GP1:90,1] + 31.571;
   1:  PR[GP1:91,2] = PR[GP1:90,2] + -37.998;
   1:L PR[91] 10mm/sec CNT100;
   1:  PR[GP1:91,1] = PR[GP1:90,1] + 43.381;
   1:  PR[GP1:91,2] = PR[GP1:90,2] + -28.649;
   1:L PR[91] 10mm/sec CNT100;
   1:  PR[GP1:91,1] = PR[GP1:90,1] + 43.862;
   1:  PR[GP1:91,2] = PR[GP1:90,2] + -28.251;
   1:L PR[91] 10mm/sec CNT100;
   1:  PR[GP1:91,1] = PR[GP1:90,1] + 51.849;
   1:  PR[GP1:91,2] = PR[GP1:90,2] + -15.027;
   1:L PR[91] 10mm/sec CNT100;
   1:  PR[GP1:91,1] = PR[GP1:90,1] + 52.040;
   1:  PR[GP1:91,2] = PR[GP1:90,2] + -13.972;
   1:L PR[91] 10mm/sec CNT100;
   1:  PR[GP1:91,1] = PR[GP1:90,1] + 52.291;
   1:  PR[GP1:91,2] = PR[GP1:90,2] + -12.415;
   1:L PR[91] 10mm/sec CNT100;
   1:  PR[GP1:91,1] = PR[GP1:90,1] + 54.577;
   1:  PR[GP1:91,2] = PR[GP1:90,2] + 0.006;
   1:L PR[91] 10mm/sec CNT100;
   1:  PR[GP1:91,1] = PR[GP1:90,1] + 54.397;
   1:  PR[GP1:91,2] = PR[GP1:90,2] + 1.207;
   1:L PR[91] 10mm/sec CNT100;
   1:  PR[GP1:91,1] = PR[GP1:90,1] + 51.850;
   1:  PR[GP1:91,2] = PR[GP1:90,2] + 15.018;
   1:L PR[91] 10mm/sec CNT100;
   1:  PR[GP1:91,1] = PR[GP1:90,1] + 43.861;
   1:  PR[GP1:91,2] = PR[GP1:90,2] + 28.244;
   1:L PR[91] 10mm/sec CNT100;
   1:  PR[GP1:91,1] = PR[GP1:90,1] + 43.380;
   1:  PR[GP1:91,2] = PR[GP1:90,2] + 28.641;
   1:L PR[91] 10mm/sec CNT100;
   1:  PR[GP1:91,1] = PR[GP1:90,1] + 31.568;
   1:  PR[GP1:91,2] = PR[GP1:90,2] + 37.991;
   1:L PR[91] 10mm/sec CNT100;
   1:  PR[GP1:91,1] = PR[GP1:90,1] + 27.266;
   1:  PR[GP1:91,2] = PR[GP1:90,2] + 39.409;
   1:L PR[91] 10mm/sec CNT100;
   1:  PR[GP1:91,1] = PR[GP1:90,1] + 16.637;
   1:  PR[GP1:91,2] = PR[GP1:90,2] + 42.986;
   1:L PR[91] 10mm/sec CNT100;
   1:  PR[GP1:91,1] = PR[GP1:90,1] + 16.335;
   1:  PR[GP1:91,2] = PR[GP1:90,2] + 43.024;
   1:L PR[91] 10mm/sec CNT100;
   1:  PR[GP1:91,1] = PR[GP1:90,1] + 1.331;
   1:  PR[GP1:91,2] = PR[GP1:90,2] + 42.636;
   1:L PR[91] 10mm/sec CNT100;
   1:  PR[GP1:91,1] = PR[GP1:90,1] + -0.458;
   1:  PR[GP1:91,2] = PR[GP1:90,2] + 42.983;
   1:  PR[GP1:91,3] = PR[GP1:90,3] + 103.740;
   1:L PR[91] 10mm/sec CNT100;
   1:  PR[GP1:91,1] = PR[GP1:90,1] + -14.704;
   1:  PR[GP1:91,2] = PR[GP1:90,2] + 43.347;
   1:L PR[91] 10mm/sec CNT100;
   1:  PR[GP1:91,1] = PR[GP1:90,1] + -15.603;
   1:  PR[GP1:91,2] = PR[GP1:90,2] + 43.235;
   1:L PR[91] 10mm/sec CNT100;
   1:  PR[GP1:91,1] = PR[GP1:90,1] + -29.986;
   1:  PR[GP1:91,2] = PR[GP1:90,2] + 38.395;
   1:L PR[91] 10mm/sec CNT100;
   1:  PR[GP1:91,1] = PR[GP1:90,1] + -30.314;
   1:  PR[GP1:91,2] = PR[GP1:90,2] + 38.268;
   1:L PR[91] 10mm/sec CNT100;
   1:  PR[GP1:91,1] = PR[GP1:90,1] + -42.639;
   1:  PR[GP1:91,2] = PR[GP1:90,2] + 28.426;
   1:L PR[91] 10mm/sec CNT100;
   1:  PR[GP1:91,1] = PR[GP1:90,1] + -50.681;
   1:  PR[GP1:91,2] = PR[GP1:90,2] + 15.118;
   1:L PR[91] 10mm/sec CNT100;
   1:  PR[GP1:91,1] = PR[GP1:90,1] + -50.830;
   1:  PR[GP1:91,2] = PR[GP1:90,2] + 14.238;
   1:L PR[91] 10mm/sec CNT100;
   1:  PR[GP1:91,1] = PR[GP1:90,1] + -53.454;
   1:  PR[GP1:91,2] = PR[GP1:90,2] + -0.015;
   1:L PR[91] 10mm/sec CNT100;
   1:  PR[GP1:91,1] = PR[GP1:90,1] + -53.381;
   1:  PR[GP1:91,2] = PR[GP1:90,2] + -0.504;
   1:L PR[91] 10mm/sec CNT100;
   1:  PR[GP1:91,1] = PR[GP1:90,1] + -50.684;
   1:  PR[GP1:91,2] = PR[GP1:90,2] + -15.123;
   1:L PR[91] 10mm/sec CNT100;
   1:  PR[GP1:91,1] = PR[GP1:90,1] + -42.640;
   1:  PR[GP1:91,2] = PR[GP1:90,2] + -28.434;
   1:L PR[91] 10mm/sec CNT100;
   1:  PR[GP1:91,1] = PR[GP1:90,1] + -30.632;
   1:  PR[GP1:91,2] = PR[GP1:90,2] + -38.057;
   1:L PR[91] 10mm/sec CNT100;
   1:  PR[GP1:91,1] = PR[GP1:90,1] + -30.333;
   1:  PR[GP1:91,2] = PR[GP1:90,2] + -38.269;
   1:L PR[91] 10mm/sec CNT100;
   1:  PR[GP1:91,1] = PR[GP1:90,1] + -29.989;
   1:  PR[GP1:91,2] = PR[GP1:90,2] + -38.402;
   1:L PR[91] 10mm/sec CNT100;
   1:  PR[GP1:91,1] = PR[GP1:90,1] + -15.607;
   1:  PR[GP1:91,2] = PR[GP1:90,2] + -43.244;
   1:L PR[91] 10mm/sec CNT100;
   1:  PR[GP1:91,1] = PR[GP1:90,1] + -14.708;
   1:  PR[GP1:91,2] = PR[GP1:90,2] + -43.355;
   1:L PR[91] 10mm/sec CNT100;
   1:  PR[GP1:91,1] = PR[GP1:90,1] + -0.458;
   1:  PR[GP1:91,2] = PR[GP1:90,2] + -42.992;
   1:L PR[91] 10mm/sec CNT100;
   1:  PR[GP1:91,1] = PR[GP1:90,1] + 1.281;
   1:L PR[91] 10mm/sec CNT100;
   1:  PR[GP1:91,1] = PR[GP1:90,1] + 15.531;
   1:  PR[GP1:91,2] = PR[GP1:90,2] + -43.355;
   1:L PR[91] 10mm/sec CNT100;
   1:  PR[GP1:91,1] = PR[GP1:90,1] + 16.430;
   1:  PR[GP1:91,2] = PR[GP1:90,2] + -43.244;
   1:L PR[91] 10mm/sec CNT100;
   1:  PR[GP1:91,1] = PR[GP1:90,1] + 30.811;
   1:  PR[GP1:91,2] = PR[GP1:90,2] + -38.402;
   1:L PR[91] 10mm/sec CNT100;
   1:  PR[GP1:91,1] = PR[GP1:90,1] + 31.139;
   1:  PR[GP1:91,2] = PR[GP1:90,2] + -38.275;
   1:L PR[91] 10mm/sec CNT100;
   1:  PR[GP1:91,1] = PR[GP1:90,1] + 43.462;
   1:  PR[GP1:91,2] = PR[GP1:90,2] + -28.430;
   1:L PR[91] 10mm/sec CNT100;
   1:  PR[GP1:91,1] = PR[GP1:90,1] + 51.502;
   1:  PR[GP1:91,2] = PR[GP1:90,2] + -15.132;
   1:L PR[91] 10mm/sec CNT100;
   1:  PR[GP1:91,1] = PR[GP1:90,1] + 51.652;
   1:  PR[GP1:91,2] = PR[GP1:90,2] + -14.250;
   1:L PR[91] 10mm/sec CNT100;
   1:  PR[GP1:91,1] = PR[GP1:90,1] + 54.275;
   1:  PR[GP1:91,2] = PR[GP1:90,2] + 0.006;
   1:L PR[91] 10mm/sec CNT100;
   1:  PR[GP1:91,1] = PR[GP1:90,1] + 54.201;
   1:  PR[GP1:91,2] = PR[GP1:90,2] + 0.496;
   1:L PR[91] 10mm/sec CNT100;
   1:  PR[GP1:91,1] = PR[GP1:90,1] + 51.504;
   1:  PR[GP1:91,2] = PR[GP1:90,2] + 15.123;
   1:L PR[91] 10mm/sec CNT100;
   1:  PR[GP1:91,1] = PR[GP1:90,1] + 51.354;
   1:  PR[GP1:91,2] = PR[GP1:90,2] + 15.375;
   1:L PR[91] 10mm/sec CNT100;
   1:  PR[GP1:91,1] = PR[GP1:90,1] + 43.461;
   1:  PR[GP1:91,2] = PR[GP1:90,2] + 28.423;
   1:L PR[91] 10mm/sec CNT100;
   1:  PR[GP1:91,1] = PR[GP1:90,1] + 31.451;
   1:  PR[GP1:91,2] = PR[GP1:90,2] + 38.050;
   1:L PR[91] 10mm/sec CNT100;
   1:  PR[GP1:91,1] = PR[GP1:90,1] + 31.153;
   1:  PR[GP1:91,2] = PR[GP1:90,2] + 38.261;
   1:L PR[91] 10mm/sec CNT100;
   1:  PR[GP1:91,1] = PR[GP1:90,1] + 30.808;
   1:  PR[GP1:91,2] = PR[GP1:90,2] + 38.394;
   1:L PR[91] 10mm/sec CNT100;
   1:  PR[GP1:91,1] = PR[GP1:90,1] + 16.426;
   1:  PR[GP1:91,2] = PR[GP1:90,2] + 43.235;
   1:L PR[91] 10mm/sec CNT100;
   1:  PR[GP1:91,1] = PR[GP1:90,1] + 15.527;
   1:  PR[GP1:91,2] = PR[GP1:90,2] + 43.347;
   1:L PR[91] 10mm/sec CNT100;
   1:  PR[GP1:91,1] = PR[GP1:90,1] + 1.281;
   1:  PR[GP1:91,2] = PR[GP1:90,2] + 42.983;
   1:L PR[91] 10mm/sec CNT100;
   1:  PR[GP1:91,1] = PR[GP1:90,1] + -0.409;
   1:  PR[GP1:91,2] = PR[GP1:90,2] + 43.330;
   1:  PR[GP1:91,3] = PR[GP1:90,3] + 105.070;
   1:L PR[91] 10mm/sec CNT100;
   1:  PR[GP1:91,1] = PR[GP1:90,1] + -11.147;
   1:  PR[GP1:91,2] = PR[GP1:90,2] + 43.610;
   1:L PR[91] 10mm/sec CNT100;
   1:  PR[GP1:91,1] = PR[GP1:90,1] + -13.894;
   1:  PR[GP1:91,2] = PR[GP1:90,2] + 43.670;
   1:L PR[91] 10mm/sec CNT100;
   1:  PR[GP1:91,1] = PR[GP1:90,1] + -15.392;
   1:  PR[GP1:91,2] = PR[GP1:90,2] + 43.484;
   1:L PR[91] 10mm/sec CNT100;
   1:  PR[GP1:91,1] = PR[GP1:90,1] + -29.004;
   1:  PR[GP1:91,2] = PR[GP1:90,2] + 38.903;
   1:L PR[91] 10mm/sec CNT100;
   1:  PR[GP1:91,1] = PR[GP1:90,1] + -29.921;
   1:  PR[GP1:91,2] = PR[GP1:90,2] + 38.548;
   1:L PR[91] 10mm/sec CNT100;
   1:  PR[GP1:91,1] = PR[GP1:90,1] + -41.714;
   1:  PR[GP1:91,2] = PR[GP1:90,2] + 29.126;
   1:L PR[91] 10mm/sec CNT100;
   1:  PR[GP1:91,1] = PR[GP1:90,1] + -42.169;
   1:  PR[GP1:91,2] = PR[GP1:90,2] + 28.803;
   1:L PR[91] 10mm/sec CNT100;
   1:  PR[GP1:91,1] = PR[GP1:90,1] + -42.534;
   1:  PR[GP1:91,2] = PR[GP1:90,2] + 28.364;
   1:L PR[91] 10mm/sec CNT100;
   1:  PR[GP1:91,1] = PR[GP1:90,1] + -50.311;
   1:  PR[GP1:91,2] = PR[GP1:90,2] + 15.372;
   1:L PR[91] 10mm/sec CNT100;
   1:  PR[GP1:91,1] = PR[GP1:90,1] + -50.399;
   1:  PR[GP1:91,2] = PR[GP1:90,2] + 15.172;
   1:L PR[91] 10mm/sec CNT100;
   1:  PR[GP1:91,1] = PR[GP1:90,1] + -53.161;
   1:  PR[GP1:91,2] = PR[GP1:90,2] + -0.004;
   1:L PR[91] 10mm/sec CNT100;
   1:  PR[GP1:91,1] = PR[GP1:90,1] + -50.429;
   1:  PR[GP1:91,2] = PR[GP1:90,2] + -14.938;
   1:L PR[91] 10mm/sec CNT100;
   1:  PR[GP1:91,1] = PR[GP1:90,1] + -50.394;
   1:  PR[GP1:91,2] = PR[GP1:90,2] + -15.191;
   1:L PR[91] 10mm/sec CNT100;
   1:  PR[GP1:91,1] = PR[GP1:90,1] + -50.311;
   1:  PR[GP1:91,2] = PR[GP1:90,2] + -15.380;
   1:L PR[91] 10mm/sec CNT100;
   1:  PR[GP1:91,1] = PR[GP1:90,1] + -42.535;
   1:  PR[GP1:91,2] = PR[GP1:90,2] + -28.371;
   1:L PR[91] 10mm/sec CNT100;
   1:  PR[GP1:91,1] = PR[GP1:90,1] + -42.159;
   1:  PR[GP1:91,2] = PR[GP1:90,2] + -28.825;
   1:L PR[91] 10mm/sec CNT100;
   1:  PR[GP1:91,1] = PR[GP1:90,1] + -30.754;
   1:  PR[GP1:91,2] = PR[GP1:90,2] + -37.973;
   1:L PR[91] 10mm/sec CNT100;
   1:  PR[GP1:91,1] = PR[GP1:90,1] + -29.940;
   1:  PR[GP1:91,2] = PR[GP1:90,2] + -38.549;
   1:L PR[91] 10mm/sec CNT100;
   1:  PR[GP1:91,1] = PR[GP1:90,1] + -29.006;
   1:  PR[GP1:91,2] = PR[GP1:90,2] + -38.911;
   1:L PR[91] 10mm/sec CNT100;
   1:  PR[GP1:91,1] = PR[GP1:90,1] + -15.396;
   1:  PR[GP1:91,2] = PR[GP1:90,2] + -43.492;
   1:L PR[91] 10mm/sec CNT100;
   1:  PR[GP1:91,1] = PR[GP1:90,1] + -13.898;
   1:  PR[GP1:91,2] = PR[GP1:90,2] + -43.678;
   1:L PR[91] 10mm/sec CNT100;
   1:  PR[GP1:91,1] = PR[GP1:90,1] + -11.141;
   1:  PR[GP1:91,2] = PR[GP1:90,2] + -43.619;
   1:L PR[91] 10mm/sec CNT100;
   1:  PR[GP1:91,1] = PR[GP1:90,1] + -0.409;
   1:  PR[GP1:91,2] = PR[GP1:90,2] + -43.339;
   1:L PR[91] 10mm/sec CNT100;
   1:  PR[GP1:91,1] = PR[GP1:90,1] + 1.232;
   1:L PR[91] 10mm/sec CNT100;
   1:  PR[GP1:91,1] = PR[GP1:90,1] + 11.964;
   1:  PR[GP1:91,2] = PR[GP1:90,2] + -43.619;
   1:L PR[91] 10mm/sec CNT100;
   1:  PR[GP1:91,1] = PR[GP1:90,1] + 14.721;
   1:  PR[GP1:91,2] = PR[GP1:90,2] + -43.678;
   1:L PR[91] 10mm/sec CNT100;
   1:  PR[GP1:91,1] = PR[GP1:90,1] + 16.219;
   1:  PR[GP1:91,2] = PR[GP1:90,2] + -43.492;
   1:L PR[91] 10mm/sec CNT100;
   1:  PR[GP1:91,1] = PR[GP1:90,1] + 29.829;
   1:  PR[GP1:91,2] = PR[GP1:90,2] + -38.910;
   1:L PR[91] 10mm/sec CNT100;
   1:  PR[GP1:91,1] = PR[GP1:90,1] + 30.746;
   1:  PR[GP1:91,2] = PR[GP1:90,2] + -38.555;
   1:L PR[91] 10mm/sec CNT100;
   1:  PR[GP1:91,1] = PR[GP1:90,1] + 42.537;
   1:  PR[GP1:91,2] = PR[GP1:90,2] + -29.130;
   1:L PR[91] 10mm/sec CNT100;
   1:  PR[GP1:91,1] = PR[GP1:90,1] + 42.992;
   1:  PR[GP1:91,2] = PR[GP1:90,2] + -28.808;
   1:L PR[91] 10mm/sec CNT100;
   1:  PR[GP1:91,1] = PR[GP1:90,1] + 43.357;
   1:  PR[GP1:91,2] = PR[GP1:90,2] + -28.368;
   1:L PR[91] 10mm/sec CNT100;
   1:  PR[GP1:91,1] = PR[GP1:90,1] + 51.132;
   1:  PR[GP1:91,2] = PR[GP1:90,2] + -15.384;
   1:L PR[91] 10mm/sec CNT100;
   1:  PR[GP1:91,1] = PR[GP1:90,1] + 51.220;
   1:  PR[GP1:91,2] = PR[GP1:90,2] + -15.185;
   1:L PR[91] 10mm/sec CNT100;
   1:  PR[GP1:91,1] = PR[GP1:90,1] + 53.982;
   1:  PR[GP1:91,2] = PR[GP1:90,2] + -0.005;
   1:L PR[91] 10mm/sec CNT100;
   1:  PR[GP1:91,1] = PR[GP1:90,1] + 51.250;
   1:  PR[GP1:91,2] = PR[GP1:90,2] + 14.935;
   1:L PR[91] 10mm/sec CNT100;
   1:  PR[GP1:91,1] = PR[GP1:90,1] + 51.215;
   1:  PR[GP1:91,2] = PR[GP1:90,2] + 15.188;
   1:L PR[91] 10mm/sec CNT100;
   1:  PR[GP1:91,1] = PR[GP1:90,1] + 51.132;
   1:  PR[GP1:91,2] = PR[GP1:90,2] + 15.377;
   1:L PR[91] 10mm/sec CNT100;
   1:  PR[GP1:91,1] = PR[GP1:90,1] + 43.356;
   1:  PR[GP1:91,2] = PR[GP1:90,2] + 28.361;
   1:L PR[91] 10mm/sec CNT100;
   1:  PR[GP1:91,1] = PR[GP1:90,1] + 42.979;
   1:  PR[GP1:91,2] = PR[GP1:90,2] + 28.814;
   1:L PR[91] 10mm/sec CNT100;
   1:  PR[GP1:91,1] = PR[GP1:90,1] + 31.573;
   1:  PR[GP1:91,2] = PR[GP1:90,2] + 37.965;
   1:L PR[91] 10mm/sec CNT100;
   1:  PR[GP1:91,1] = PR[GP1:90,1] + 30.760;
   1:  PR[GP1:91,2] = PR[GP1:90,2] + 38.541;
   1:L PR[91] 10mm/sec CNT100;
   1:  PR[GP1:91,1] = PR[GP1:90,1] + 29.826;
   1:  PR[GP1:91,2] = PR[GP1:90,2] + 38.903;
   1:L PR[91] 10mm/sec CNT100;
   1:  PR[GP1:91,1] = PR[GP1:90,1] + 16.215;
   1:  PR[GP1:91,2] = PR[GP1:90,2] + 43.484;
   1:L PR[91] 10mm/sec CNT100;
   1:  PR[GP1:91,1] = PR[GP1:90,1] + 14.717;
   1:  PR[GP1:91,2] = PR[GP1:90,2] + 43.669;
   1:L PR[91] 10mm/sec CNT100;
   1:  PR[GP1:91,1] = PR[GP1:90,1] + 11.970;
   1:  PR[GP1:91,2] = PR[GP1:90,2] + 43.610;
   1:L PR[91] 10mm/sec CNT100;
   1:  PR[GP1:91,1] = PR[GP1:90,1] + 1.232;
   1:  PR[GP1:91,2] = PR[GP1:90,2] + 43.330;
   1:L PR[91] 10mm/sec CNT100;
   1:  PR[GP1:91,1] = PR[GP1:90,1] + -0.360;
   1:  PR[GP1:91,2] = PR[GP1:90,2] + 43.678;
   1:  PR[GP1:91,3] = PR[GP1:90,3] + 106.400;
   1:L PR[91] 10mm/sec CNT100;
   1:  PR[GP1:91,1] = PR[GP1:90,1] + -9.297;
   1:  PR[GP1:91,2] = PR[GP1:90,2] + 43.911;
   1:L PR[91] 10mm/sec CNT100;
   1:  PR[GP1:91,1] = PR[GP1:90,1] + -13.087;
   1:  PR[GP1:91,2] = PR[GP1:90,2] + 43.992;
   1:L PR[91] 10mm/sec CNT100;
   1:  PR[GP1:91,1] = PR[GP1:90,1] + -15.182;
   1:  PR[GP1:91,2] = PR[GP1:90,2] + 43.733;
   1:L PR[91] 10mm/sec CNT100;
   1:  PR[GP1:91,1] = PR[GP1:90,1] + -28.022;
   1:  PR[GP1:91,2] = PR[GP1:90,2] + 39.411;
   1:L PR[91] 10mm/sec CNT100;
   1:  PR[GP1:91,1] = PR[GP1:90,1] + -29.528;
   1:  PR[GP1:91,2] = PR[GP1:90,2] + 38.828;
   1:L PR[91] 10mm/sec CNT100;
   1:  PR[GP1:91,1] = PR[GP1:90,1] + -40.652;
   1:  PR[GP1:91,2] = PR[GP1:90,2] + 29.939;
   1:L PR[91] 10mm/sec CNT100;
   1:  PR[GP1:91,1] = PR[GP1:90,1] + -41.645;
   1:  PR[GP1:91,2] = PR[GP1:90,2] + 29.237;
   1:L PR[91] 10mm/sec CNT100;
   1:  PR[GP1:91,1] = PR[GP1:90,1] + -42.482;
   1:  PR[GP1:91,2] = PR[GP1:90,2] + 28.228;
   1:L PR[91] 10mm/sec CNT100;
   1:  PR[GP1:91,1] = PR[GP1:90,1] + -49.818;
   1:  PR[GP1:91,2] = PR[GP1:90,2] + 15.973;
   1:L PR[91] 10mm/sec CNT100;
   1:  PR[GP1:91,1] = PR[GP1:90,1] + -50.213;
   1:  PR[GP1:91,2] = PR[GP1:90,2] + 15.078;
   1:L PR[91] 10mm/sec CNT100;
   1:  PR[GP1:91,1] = PR[GP1:90,1] + -52.819;
   1:  PR[GP1:91,2] = PR[GP1:90,2] + 0.785;
   1:L PR[91] 10mm/sec CNT100;
   1:  PR[GP1:91,1] = PR[GP1:90,1] + -52.928;
   1:  PR[GP1:91,2] = PR[GP1:90,2] + 0.008;
   1:L PR[91] 10mm/sec CNT100;
   1:  PR[GP1:91,1] = PR[GP1:90,1] + -50.349;
   1:  PR[GP1:91,2] = PR[GP1:90,2] + -14.091;
   1:L PR[91] 10mm/sec CNT100;
   1:  PR[GP1:91,1] = PR[GP1:90,1] + -50.208;
   1:  PR[GP1:91,2] = PR[GP1:90,2] + -15.097;
   1:L PR[91] 10mm/sec CNT100;
   1:  PR[GP1:91,1] = PR[GP1:90,1] + -49.818;
   1:  PR[GP1:91,2] = PR[GP1:90,2] + -15.981;
   1:L PR[91] 10mm/sec CNT100;
   1:  PR[GP1:91,1] = PR[GP1:90,1] + -42.483;
   1:  PR[GP1:91,2] = PR[GP1:90,2] + -28.236;
   1:L PR[91] 10mm/sec CNT100;
   1:  PR[GP1:91,1] = PR[GP1:90,1] + -41.634;
   1:  PR[GP1:91,2] = PR[GP1:90,2] + -29.258;
   1:L PR[91] 10mm/sec CNT100;
   1:  PR[GP1:91,1] = PR[GP1:90,1] + -30.876;
   1:  PR[GP1:91,2] = PR[GP1:90,2] + -37.888;
   1:L PR[91] 10mm/sec CNT100;
   1:  PR[GP1:91,1] = PR[GP1:90,1] + -29.547;
   1:  PR[GP1:91,2] = PR[GP1:90,2] + -38.829;
   1:L PR[91] 10mm/sec CNT100;
   1:  PR[GP1:91,1] = PR[GP1:90,1] + -28.025;
   1:  PR[GP1:91,2] = PR[GP1:90,2] + -39.419;
   1:L PR[91] 10mm/sec CNT100;
   1:  PR[GP1:91,1] = PR[GP1:90,1] + -15.185;
   1:  PR[GP1:91,2] = PR[GP1:90,2] + -43.741;
   1:L PR[91] 10mm/sec CNT100;
   1:  PR[GP1:91,1] = PR[GP1:90,1] + -13.090;
   1:  PR[GP1:91,2] = PR[GP1:90,2] + -44.001;
   1:L PR[91] 10mm/sec CNT100;
   1:  PR[GP1:91,1] = PR[GP1:90,1] + -9.287;
   1:  PR[GP1:91,2] = PR[GP1:90,2] + -43.919;
   1:L PR[91] 10mm/sec CNT100;
   1:  PR[GP1:91,1] = PR[GP1:90,1] + -0.360;
   1:  PR[GP1:91,2] = PR[GP1:90,2] + -43.687;
   1:L PR[91] 10mm/sec CNT100;
   1:  PR[GP1:91,1] = PR[GP1:90,1] + 1.182;
   1:L PR[91] 10mm/sec CNT100;
   1:  PR[GP1:91,1] = PR[GP1:90,1] + 10.110;
   1:  PR[GP1:91,2] = PR[GP1:90,2] + -43.919;
   1:L PR[91] 10mm/sec CNT100;
   1:  PR[GP1:91,1] = PR[GP1:90,1] + 13.912;
   1:  PR[GP1:91,2] = PR[GP1:90,2] + -44.001;
   1:L PR[91] 10mm/sec CNT100;
   1:  PR[GP1:91,1] = PR[GP1:90,1] + 16.008;
   1:  PR[GP1:91,2] = PR[GP1:90,2] + -43.741;
   1:L PR[91] 10mm/sec CNT100;
   1:  PR[GP1:91,1] = PR[GP1:90,1] + 28.847;
   1:  PR[GP1:91,2] = PR[GP1:90,2] + -39.418;
   1:L PR[91] 10mm/sec CNT100;
   1:  PR[GP1:91,1] = PR[GP1:90,1] + 30.353;
   1:  PR[GP1:91,2] = PR[GP1:90,2] + -38.835;
   1:L PR[91] 10mm/sec CNT100;
   1:  PR[GP1:91,1] = PR[GP1:90,1] + 41.475;
   1:  PR[GP1:91,2] = PR[GP1:90,2] + -29.944;
   1:L PR[91] 10mm/sec CNT100;
   1:  PR[GP1:91,1] = PR[GP1:90,1] + 42.468;
   1:  PR[GP1:91,2] = PR[GP1:90,2] + -29.241;
   1:L PR[91] 10mm/sec CNT100;
   1:  PR[GP1:91,1] = PR[GP1:90,1] + 43.305;
   1:  PR[GP1:91,2] = PR[GP1:90,2] + -28.233;
   1:L PR[91] 10mm/sec CNT100;
   1:  PR[GP1:91,1] = PR[GP1:90,1] + 50.639;
   1:  PR[GP1:91,2] = PR[GP1:90,2] + -15.985;
   1:L PR[91] 10mm/sec CNT100;
   1:  PR[GP1:91,1] = PR[GP1:90,1] + 51.034;
   1:  PR[GP1:91,2] = PR[GP1:90,2] + -15.090;
   1:L PR[91] 10mm/sec CNT100;
   1:  PR[GP1:91,1] = PR[GP1:90,1] + 53.640;
   1:  PR[GP1:91,2] = PR[GP1:90,2] + -0.793;
   1:L PR[91] 10mm/sec CNT100;
   1:  PR[GP1:91,1] = PR[GP1:90,1] + 53.748;
   1:  PR[GP1:91,2] = PR[GP1:90,2] + -0.017;
   1:L PR[91] 10mm/sec CNT100;
   1:  PR[GP1:91,1] = PR[GP1:90,1] + 51.169;
   1:  PR[GP1:91,2] = PR[GP1:90,2] + 14.088;
   1:L PR[91] 10mm/sec CNT100;
   1:  PR[GP1:91,1] = PR[GP1:90,1] + 51.029;
   1:  PR[GP1:91,2] = PR[GP1:90,2] + 15.094;
   1:L PR[91] 10mm/sec CNT100;
   1:  PR[GP1:91,1] = PR[GP1:90,1] + 50.639;
   1:  PR[GP1:91,2] = PR[GP1:90,2] + 15.977;
   1:L PR[91] 10mm/sec CNT100;
   1:  PR[GP1:91,1] = PR[GP1:90,1] + 43.304;
   1:  PR[GP1:91,2] = PR[GP1:90,2] + 28.226;
   1:L PR[91] 10mm/sec CNT100;
   1:  PR[GP1:91,1] = PR[GP1:90,1] + 42.455;
   1:  PR[GP1:91,2] = PR[GP1:90,2] + 29.248;
   1:L PR[91] 10mm/sec CNT100;
   1:  PR[GP1:91,1] = PR[GP1:90,1] + 31.696;
   1:  PR[GP1:91,2] = PR[GP1:90,2] + 37.880;
   1:L PR[91] 10mm/sec CNT100;
   1:  PR[GP1:91,1] = PR[GP1:90,1] + 30.367;
   1:  PR[GP1:91,2] = PR[GP1:90,2] + 38.821;
   1:L PR[91] 10mm/sec CNT100;
   1:  PR[GP1:91,1] = PR[GP1:90,1] + 28.844;
   1:  PR[GP1:91,2] = PR[GP1:90,2] + 39.411;
   1:L PR[91] 10mm/sec CNT100;
   1:  PR[GP1:91,1] = PR[GP1:90,1] + 16.004;
   1:  PR[GP1:91,2] = PR[GP1:90,2] + 43.733;
   1:L PR[91] 10mm/sec CNT100;
   1:  PR[GP1:91,1] = PR[GP1:90,1] + 13.909;
   1:  PR[GP1:91,2] = PR[GP1:90,2] + 43.992;
   1:L PR[91] 10mm/sec CNT100;
   1:  PR[GP1:91,1] = PR[GP1:90,1] + 10.119;
   1:  PR[GP1:91,2] = PR[GP1:90,2] + 43.911;
   1:L PR[91] 10mm/sec CNT100;
   1:  PR[GP1:91,1] = PR[GP1:90,1] + 1.182;
   1:  PR[GP1:91,2] = PR[GP1:90,2] + 43.678;
   1:L PR[91] 10mm/sec CNT100;
   1:  PR[GP1:91,1] = PR[GP1:90,1] + -0.311;
   1:  PR[GP1:91,2] = PR[GP1:90,2] + 44.025;
   1:  PR[GP1:91,3] = PR[GP1:90,3] + 107.730;
   1:L PR[91] 10mm/sec CNT100;
   1:  PR[GP1:91,1] = PR[GP1:90,1] + -7.446;
   1:  PR[GP1:91,2] = PR[GP1:90,2] + 44.211;
   1:L PR[91] 10mm/sec CNT100;
   1:  PR[GP1:91,1] = PR[GP1:90,1] + -12.279;
   1:  PR[GP1:91,2] = PR[GP1:90,2] + 44.315;
   1:L PR[91] 10mm/sec CNT100;
   1:  PR[GP1:91,1] = PR[GP1:90,1] + -14.971;
   1:  PR[GP1:91,2] = PR[GP1:90,2] + 43.981;
   1:L PR[91] 10mm/sec CNT100;
   1:  PR[GP1:91,1] = PR[GP1:90,1] + -27.040;
   1:  PR[GP1:91,2] = PR[GP1:90,2] + 39.920;
   1:L PR[91] 10mm/sec CNT100;
   1:  PR[GP1:91,1] = PR[GP1:90,1] + -29.135;
   1:  PR[GP1:91,2] = PR[GP1:90,2] + 39.108;
   1:L PR[91] 10mm/sec CNT100;
   1:  PR[GP1:91,1] = PR[GP1:90,1] + -39.591;
   1:  PR[GP1:91,2] = PR[GP1:90,2] + 30.753;
   1:L PR[91] 10mm/sec CNT100;
   1:  PR[GP1:91,1] = PR[GP1:90,1] + -41.121;
   1:  PR[GP1:91,2] = PR[GP1:90,2] + 29.671;
   1:L PR[91] 10mm/sec CNT100;
   1:  PR[GP1:91,1] = PR[GP1:90,1] + -42.430;
   1:  PR[GP1:91,2] = PR[GP1:90,2] + 28.093;
   1:L PR[91] 10mm/sec CNT100;
   1:  PR[GP1:91,1] = PR[GP1:90,1] + -49.325;
   1:  PR[GP1:91,2] = PR[GP1:90,2] + 16.574;
   1:L PR[91] 10mm/sec CNT100;
   1:  PR[GP1:91,1] = PR[GP1:90,1] + -50.027;
   1:  PR[GP1:91,2] = PR[GP1:90,2] + 14.983;
   1:L PR[91] 10mm/sec CNT100;
   1:  PR[GP1:91,1] = PR[GP1:90,1] + -52.477;
   1:  PR[GP1:91,2] = PR[GP1:90,2] + 1.549;
   1:L PR[91] 10mm/sec CNT100;
   1:  PR[GP1:91,1] = PR[GP1:90,1] + -52.692;
   1:  PR[GP1:91,2] = PR[GP1:90,2] + 0.008;
   1:L PR[91] 10mm/sec CNT100;
   1:  PR[GP1:91,1] = PR[GP1:90,1] + -50.268;
   1:  PR[GP1:91,2] = PR[GP1:90,2] + -13.244;
   1:L PR[91] 10mm/sec CNT100;
   1:  PR[GP1:91,1] = PR[GP1:90,1] + -50.023;
   1:  PR[GP1:91,2] = PR[GP1:90,2] + -15.003;
   1:L PR[91] 10mm/sec CNT100;
   1:  PR[GP1:91,1] = PR[GP1:90,1] + -49.325;
   1:  PR[GP1:91,2] = PR[GP1:90,2] + -16.582;
   1:L PR[91] 10mm/sec CNT100;
   1:  PR[GP1:91,1] = PR[GP1:90,1] + -42.431;
   1:  PR[GP1:91,2] = PR[GP1:90,2] + -28.101;
   1:L PR[91] 10mm/sec CNT100;
   1:  PR[GP1:91,1] = PR[GP1:90,1] + -41.110;
   1:  PR[GP1:91,2] = PR[GP1:90,2] + -29.692;
   1:L PR[91] 10mm/sec CNT100;
   1:  PR[GP1:91,1] = PR[GP1:90,1] + -30.998;
   1:  PR[GP1:91,2] = PR[GP1:90,2] + -37.803;
   1:L PR[91] 10mm/sec CNT100;
   1:  PR[GP1:91,1] = PR[GP1:90,1] + -29.154;
   1:  PR[GP1:91,2] = PR[GP1:90,2] + -39.109;
   1:L PR[91] 10mm/sec CNT100;
   1:  PR[GP1:91,1] = PR[GP1:90,1] + -27.043;
   1:  PR[GP1:91,2] = PR[GP1:90,2] + -39.927;
   1:L PR[91] 10mm/sec CNT100;
   1:  PR[GP1:91,1] = PR[GP1:90,1] + -14.974;
   1:  PR[GP1:91,2] = PR[GP1:90,2] + -43.990;
   1:L PR[91] 10mm/sec CNT100;
   1:  PR[GP1:91,1] = PR[GP1:90,1] + -12.282;
   1:  PR[GP1:91,2] = PR[GP1:90,2] + -44.323;
   1:L PR[91] 10mm/sec CNT100;
   1:  PR[GP1:91,1] = PR[GP1:90,1] + -7.433;
   1:  PR[GP1:91,2] = PR[GP1:90,2] + -44.219;
   1:L PR[91] 10mm/sec CNT100;
   1:  PR[GP1:91,1] = PR[GP1:90,1] + -0.311;
   1:  PR[GP1:91,2] = PR[GP1:90,2] + -44.034;
   1:L PR[91] 10mm/sec CNT100;
   1:  PR[GP1:91,1] = PR[GP1:90,1] + 1.133;
   1:L PR[91] 10mm/sec CNT100;
   1:  PR[GP1:91,1] = PR[GP1:90,1] + 8.255;
   1:  PR[GP1:91,2] = PR[GP1:90,2] + -44.219;
   1:L PR[91] 10mm/sec CNT100;
   1:  PR[GP1:91,1] = PR[GP1:90,1] + 13.104;
   1:  PR[GP1:91,2] = PR[GP1:90,2] + -44.323;
   1:L PR[91] 10mm/sec CNT100;
   1:  PR[GP1:91,1] = PR[GP1:90,1] + 15.796;
   1:  PR[GP1:91,2] = PR[GP1:90,2] + -43.990;
   1:L PR[91] 10mm/sec CNT100;
   1:  PR[GP1:91,1] = PR[GP1:90,1] + 27.865;
   1:  PR[GP1:91,2] = PR[GP1:90,2] + -39.927;
   1:L PR[91] 10mm/sec CNT100;
   1:  PR[GP1:91,1] = PR[GP1:90,1] + 29.959;
   1:  PR[GP1:91,2] = PR[GP1:90,2] + -39.115;
   1:L PR[91] 10mm/sec CNT100;
   1:  PR[GP1:91,1] = PR[GP1:90,1] + 40.414;
   1:  PR[GP1:91,2] = PR[GP1:90,2] + -30.758;
   1:L PR[91] 10mm/sec CNT100;
   1:  PR[GP1:91,1] = PR[GP1:90,1] + 41.943;
   1:  PR[GP1:91,2] = PR[GP1:90,2] + -29.675;
   1:L PR[91] 10mm/sec CNT100;
   1:  PR[GP1:91,1] = PR[GP1:90,1] + 43.253;
   1:  PR[GP1:91,2] = PR[GP1:90,2] + -28.098;
   1:L PR[91] 10mm/sec CNT100;
   1:  PR[GP1:91,1] = PR[GP1:90,1] + 50.146;
   1:  PR[GP1:91,2] = PR[GP1:90,2] + -16.586;
   1:L PR[91] 10mm/sec CNT100;
   1:  PR[GP1:91,1] = PR[GP1:90,1] + 50.849;
   1:  PR[GP1:91,2] = PR[GP1:90,2] + -14.996;
   1:L PR[91] 10mm/sec CNT100;
   1:  PR[GP1:91,1] = PR[GP1:90,1] + 53.298;
   1:  PR[GP1:91,2] = PR[GP1:90,2] + -1.558;
   1:L PR[91] 10mm/sec CNT100;
   1:  PR[GP1:91,1] = PR[GP1:90,1] + 53.512;
   1:  PR[GP1:91,2] = PR[GP1:90,2] + -0.017;
   1:L PR[91] 10mm/sec CNT100;
   1:  PR[GP1:91,1] = PR[GP1:90,1] + 51.089;
   1:  PR[GP1:91,2] = PR[GP1:90,2] + 13.240;
   1:L PR[91] 10mm/sec CNT100;
   1:  PR[GP1:91,1] = PR[GP1:90,1] + 50.843;
   1:  PR[GP1:91,2] = PR[GP1:90,2] + 14.999;
   1:L PR[91] 10mm/sec CNT100;
   1:  PR[GP1:91,1] = PR[GP1:90,1] + 50.146;
   1:  PR[GP1:91,2] = PR[GP1:90,2] + 16.578;
   1:L PR[91] 10mm/sec CNT100;
   1:  PR[GP1:91,1] = PR[GP1:90,1] + 43.252;
   1:  PR[GP1:91,2] = PR[GP1:90,2] + 28.091;
   1:L PR[91] 10mm/sec CNT100;
   1:  PR[GP1:91,1] = PR[GP1:90,1] + 41.931;
   1:  PR[GP1:91,2] = PR[GP1:90,2] + 29.682;
   1:L PR[91] 10mm/sec CNT100;
   1:  PR[GP1:91,1] = PR[GP1:90,1] + 31.818;
   1:  PR[GP1:91,2] = PR[GP1:90,2] + 37.795;
   1:L PR[91] 10mm/sec CNT100;
   1:  PR[GP1:91,1] = PR[GP1:90,1] + 29.974;
   1:  PR[GP1:91,2] = PR[GP1:90,2] + 39.101;
   1:L PR[91] 10mm/sec CNT100;
   1:  PR[GP1:91,1] = PR[GP1:90,1] + 27.862;
   1:  PR[GP1:91,2] = PR[GP1:90,2] + 39.919;
   1:L PR[91] 10mm/sec CNT100;
   1:  PR[GP1:91,1] = PR[GP1:90,1] + 15.793;
   1:  PR[GP1:91,2] = PR[GP1:90,2] + 43.981;
   1:L PR[91] 10mm/sec CNT100;
   1:  PR[GP1:91,1] = PR[GP1:90,1] + 13.101;
   1:  PR[GP1:91,2] = PR[GP1:90,2] + 44.315;
   1:L PR[91] 10mm/sec CNT100;
   1:  PR[GP1:91,1] = PR[GP1:90,1] + 8.268;
   1:  PR[GP1:91,2] = PR[GP1:90,2] + 44.211;
   1:L PR[91] 10mm/sec CNT100;
   1:  PR[GP1:91,1] = PR[GP1:90,1] + 1.133;
   1:  PR[GP1:91,2] = PR[GP1:90,2] + 44.025;
   1:L PR[91] 10mm/sec CNT100;
   1:  PR[GP1:91,1] = PR[GP1:90,1] + -0.262;
   1:  PR[GP1:91,2] = PR[GP1:90,2] + 44.372;
   1:  PR[GP1:91,3] = PR[GP1:90,3] + 109.060;
   1:L PR[91] 10mm/sec CNT100;
   1:  PR[GP1:91,1] = PR[GP1:90,1] + -5.596;
   1:  PR[GP1:91,2] = PR[GP1:90,2] + 44.511;
   1:L PR[91] 10mm/sec CNT100;
   1:  PR[GP1:91,1] = PR[GP1:90,1] + -11.471;
   1:  PR[GP1:91,2] = PR[GP1:90,2] + 44.638;
   1:L PR[91] 10mm/sec CNT100;
   1:  PR[GP1:91,1] = PR[GP1:90,1] + -14.761;
   1:  PR[GP1:91,2] = PR[GP1:90,2] + 44.230;
   1:L PR[91] 10mm/sec CNT100;
   1:  PR[GP1:91,1] = PR[GP1:90,1] + -26.059;
   1:  PR[GP1:91,2] = PR[GP1:90,2] + 40.428;
   1:L PR[91] 10mm/sec CNT100;
   1:  PR[GP1:91,1] = PR[GP1:90,1] + -28.742;
   1:  PR[GP1:91,2] = PR[GP1:90,2] + 39.388;
   1:L PR[91] 10mm/sec CNT100;
   1:  PR[GP1:91,1] = PR[GP1:90,1] + -38.530;
   1:  PR[GP1:91,2] = PR[GP1:90,2] + 31.567;
   1:L PR[91] 10mm/sec CNT100;
   1:  PR[GP1:91,1] = PR[GP1:90,1] + -40.596;
   1:  PR[GP1:91,2] = PR[GP1:90,2] + 30.104;
   1:L PR[91] 10mm/sec CNT100;
   1:  PR[GP1:91,1] = PR[GP1:90,1] + -42.378;
   1:  PR[GP1:91,2] = PR[GP1:90,2] + 27.958;
   1:L PR[91] 10mm/sec CNT100;
   1:  PR[GP1:91,1] = PR[GP1:90,1] + -48.832;
   1:  PR[GP1:91,2] = PR[GP1:90,2] + 17.175;
   1:L PR[91] 10mm/sec CNT100;
   1:  PR[GP1:91,1] = PR[GP1:90,1] + -49.842;
   1:  PR[GP1:91,2] = PR[GP1:90,2] + 14.889;
   1:L PR[91] 10mm/sec CNT100;
   1:  PR[GP1:91,1] = PR[GP1:90,1] + -52.135;
   1:  PR[GP1:91,2] = PR[GP1:90,2] + 2.314;
   1:L PR[91] 10mm/sec CNT100;
   1:  PR[GP1:91,1] = PR[GP1:90,1] + -52.456;
   1:  PR[GP1:91,2] = PR[GP1:90,2] + 0.008;
   1:L PR[91] 10mm/sec CNT100;
   1:  PR[GP1:91,1] = PR[GP1:90,1] + -50.187;
   1:  PR[GP1:91,2] = PR[GP1:90,2] + -12.397;
   1:L PR[91] 10mm/sec CNT100;
   1:  PR[GP1:91,1] = PR[GP1:90,1] + -49.837;
   1:  PR[GP1:91,2] = PR[GP1:90,2] + -14.909;
   1:L PR[91] 10mm/sec CNT100;
   1:  PR[GP1:91,1] = PR[GP1:90,1] + -48.833;
   1:  PR[GP1:91,2] = PR[GP1:90,2] + -17.184;
   1:L PR[91] 10mm/sec CNT100;
   1:  PR[GP1:91,1] = PR[GP1:90,1] + -42.379;
   1:  PR[GP1:91,2] = PR[GP1:90,2] + -27.966;
   1:L PR[91] 10mm/sec CNT100;
   1:  PR[GP1:91,1] = PR[GP1:90,1] + -40.586;
   1:  PR[GP1:91,2] = PR[GP1:90,2] + -30.126;
   1:L PR[91] 10mm/sec CNT100;
   1:  PR[GP1:91,1] = PR[GP1:90,1] + -31.120;
   1:  PR[GP1:91,2] = PR[GP1:90,2] + -37.719;
   1:L PR[91] 10mm/sec CNT100;
   1:  PR[GP1:91,1] = PR[GP1:90,1] + -28.760;
   1:  PR[GP1:91,2] = PR[GP1:90,2] + -39.389;
   1:L PR[91] 10mm/sec CNT100;
   1:  PR[GP1:91,1] = PR[GP1:90,1] + -26.061;
   1:  PR[GP1:91,2] = PR[GP1:90,2] + -40.436;
   1:L PR[91] 10mm/sec CNT100;
   1:  PR[GP1:91,1] = PR[GP1:90,1] + -14.764;
   1:  PR[GP1:91,2] = PR[GP1:90,2] + -44.239;
   1:L PR[91] 10mm/sec CNT100;
   1:  PR[GP1:91,1] = PR[GP1:90,1] + -11.474;
   1:  PR[GP1:91,2] = PR[GP1:90,2] + -44.646;
   1:L PR[91] 10mm/sec CNT100;
   1:  PR[GP1:91,1] = PR[GP1:90,1] + -5.580;
   1:  PR[GP1:91,2] = PR[GP1:90,2] + -44.520;
   1:L PR[91] 10mm/sec CNT100;
   1:  PR[GP1:91,1] = PR[GP1:90,1] + -0.262;
   1:  PR[GP1:91,2] = PR[GP1:90,2] + -44.381;
   1:L PR[91] 10mm/sec CNT100;
   1:  PR[GP1:91,1] = PR[GP1:90,1] + 1.083;
   1:L PR[91] 10mm/sec CNT100;
   1:  PR[GP1:91,1] = PR[GP1:90,1] + 6.401;
   1:  PR[GP1:91,2] = PR[GP1:90,2] + -44.519;
   1:L PR[91] 10mm/sec CNT100;
   1:  PR[GP1:91,1] = PR[GP1:90,1] + 12.295;
   1:  PR[GP1:91,2] = PR[GP1:90,2] + -44.646;
   1:L PR[91] 10mm/sec CNT100;
   1:  PR[GP1:91,1] = PR[GP1:90,1] + 15.585;
   1:  PR[GP1:91,2] = PR[GP1:90,2] + -44.239;
   1:L PR[91] 10mm/sec CNT100;
   1:  PR[GP1:91,1] = PR[GP1:90,1] + 26.883;
   1:  PR[GP1:91,2] = PR[GP1:90,2] + -40.435;
   1:L PR[91] 10mm/sec CNT100;
   1:  PR[GP1:91,1] = PR[GP1:90,1] + 29.566;
   1:  PR[GP1:91,2] = PR[GP1:90,2] + -39.395;
   1:L PR[91] 10mm/sec CNT100;
   1:  PR[GP1:91,1] = PR[GP1:90,1] + 39.353;
   1:  PR[GP1:91,2] = PR[GP1:90,2] + -31.572;
   1:L PR[91] 10mm/sec CNT100;
   1:  PR[GP1:91,1] = PR[GP1:90,1] + 41.419;
   1:  PR[GP1:91,2] = PR[GP1:90,2] + -30.109;
   1:L PR[91] 10mm/sec CNT100;
   1:  PR[GP1:91,1] = PR[GP1:90,1] + 43.201;
   1:  PR[GP1:91,2] = PR[GP1:90,2] + -27.963;
   1:L PR[91] 10mm/sec CNT100;
   1:  PR[GP1:91,1] = PR[GP1:90,1] + 49.654;
   1:  PR[GP1:91,2] = PR[GP1:90,2] + -17.187;
   1:L PR[91] 10mm/sec CNT100;
   1:  PR[GP1:91,1] = PR[GP1:90,1] + 50.663;
   1:  PR[GP1:91,2] = PR[GP1:90,2] + -14.901;
   1:L PR[91] 10mm/sec CNT100;
   1:  PR[GP1:91,1] = PR[GP1:90,1] + 52.955;
   1:  PR[GP1:91,2] = PR[GP1:90,2] + -2.322;
   1:L PR[91] 10mm/sec CNT100;
   1:  PR[GP1:91,1] = PR[GP1:90,1] + 53.277;
   1:  PR[GP1:91,2] = PR[GP1:90,2] + -0.017;
   1:L PR[91] 10mm/sec CNT100;
   1:  PR[GP1:91,1] = PR[GP1:90,1] + 51.008;
   1:  PR[GP1:91,2] = PR[GP1:90,2] + 12.393;
   1:L PR[91] 10mm/sec CNT100;
   1:  PR[GP1:91,1] = PR[GP1:90,1] + 50.657;
   1:  PR[GP1:91,2] = PR[GP1:90,2] + 14.905;
   1:L PR[91] 10mm/sec CNT100;
   1:  PR[GP1:91,1] = PR[GP1:90,1] + 49.653;
   1:  PR[GP1:91,2] = PR[GP1:90,2] + 17.179;
   1:L PR[91] 10mm/sec CNT100;
   1:  PR[GP1:91,1] = PR[GP1:90,1] + 43.200;
   1:  PR[GP1:91,2] = PR[GP1:90,2] + 27.956;
   1:L PR[91] 10mm/sec CNT100;
   1:  PR[GP1:91,1] = PR[GP1:90,1] + 41.406;
   1:  PR[GP1:91,2] = PR[GP1:90,2] + 30.115;
   1:L PR[91] 10mm/sec CNT100;
   1:  PR[GP1:91,1] = PR[GP1:90,1] + 31.940;
   1:  PR[GP1:91,2] = PR[GP1:90,2] + 37.710;
   1:L PR[91] 10mm/sec CNT100;
   1:  PR[GP1:91,1] = PR[GP1:90,1] + 29.580;
   1:  PR[GP1:91,2] = PR[GP1:90,2] + 39.381;
   1:L PR[91] 10mm/sec CNT100;
   1:  PR[GP1:91,1] = PR[GP1:90,1] + 26.880;
   1:  PR[GP1:91,2] = PR[GP1:90,2] + 40.428;
   1:L PR[91] 10mm/sec CNT100;
   1:  PR[GP1:91,1] = PR[GP1:90,1] + 15.583;
   1:  PR[GP1:91,2] = PR[GP1:90,2] + 44.230;
   1:L PR[91] 10mm/sec CNT100;
   1:  PR[GP1:91,1] = PR[GP1:90,1] + 12.292;
   1:  PR[GP1:91,2] = PR[GP1:90,2] + 44.638;
   1:L PR[91] 10mm/sec CNT100;
   1:  PR[GP1:91,1] = PR[GP1:90,1] + 6.418;
   1:  PR[GP1:91,2] = PR[GP1:90,2] + 44.511;
   1:L PR[91] 10mm/sec CNT100;
   1:  PR[GP1:91,1] = PR[GP1:90,1] + 1.083;
   1:  PR[GP1:91,2] = PR[GP1:90,2] + 44.372;
   1:L PR[91] 10mm/sec CNT100;
   1:  PR[GP1:91,1] = PR[GP1:90,1] + -0.213;
   1:  PR[GP1:91,2] = PR[GP1:90,2] + 44.719;
   1:  PR[GP1:91,3] = PR[GP1:90,3] + 110.390;
   1:L PR[91] 10mm/sec CNT100;
   1:  PR[GP1:91,1] = PR[GP1:90,1] + -3.746;
   1:  PR[GP1:91,2] = PR[GP1:90,2] + 44.812;
   1:L PR[91] 10mm/sec CNT100;
   1:  PR[GP1:91,1] = PR[GP1:90,1] + -10.663;
   1:  PR[GP1:91,2] = PR[GP1:90,2] + 44.960;
   1:L PR[91] 10mm/sec CNT100;
   1:  PR[GP1:91,1] = PR[GP1:90,1] + -14.550;
   1:  PR[GP1:91,2] = PR[GP1:90,2] + 44.479;
   1:L PR[91] 10mm/sec CNT100;
   1:  PR[GP1:91,1] = PR[GP1:90,1] + -25.077;
   1:  PR[GP1:91,2] = PR[GP1:90,2] + 40.936;
   1:L PR[91] 10mm/sec CNT100;
   1:  PR[GP1:91,1] = PR[GP1:90,1] + -28.349;
   1:  PR[GP1:91,2] = PR[GP1:90,2] + 39.668;
   1:L PR[91] 10mm/sec CNT100;
   1:  PR[GP1:91,1] = PR[GP1:90,1] + -37.469;
   1:  PR[GP1:91,2] = PR[GP1:90,2] + 32.381;
   1:L PR[91] 10mm/sec CNT100;
   1:  PR[GP1:91,1] = PR[GP1:90,1] + -40.072;
   1:  PR[GP1:91,2] = PR[GP1:90,2] + 30.538;
   1:L PR[91] 10mm/sec CNT100;
   1:  PR[GP1:91,1] = PR[GP1:90,1] + -42.326;
   1:  PR[GP1:91,2] = PR[GP1:90,2] + 27.823;
   1:L PR[91] 10mm/sec CNT100;
   1:  PR[GP1:91,1] = PR[GP1:90,1] + -48.340;
   1:  PR[GP1:91,2] = PR[GP1:90,2] + 17.777;
   1:L PR[91] 10mm/sec CNT100;
   1:  PR[GP1:91,1] = PR[GP1:90,1] + -49.656;
   1:  PR[GP1:91,2] = PR[GP1:90,2] + 14.795;
   1:L PR[91] 10mm/sec CNT100;
   1:  PR[GP1:91,1] = PR[GP1:90,1] + -51.792;
   1:  PR[GP1:91,2] = PR[GP1:90,2] + 3.078;
   1:L PR[91] 10mm/sec CNT100;
   1:  PR[GP1:91,1] = PR[GP1:90,1] + -52.220;
   1:  PR[GP1:91,2] = PR[GP1:90,2] + 0.008;
   1:L PR[91] 10mm/sec CNT100;
   1:  PR[GP1:91,1] = PR[GP1:90,1] + -50.107;
   1:  PR[GP1:91,2] = PR[GP1:90,2] + -11.550;
   1:L PR[91] 10mm/sec CNT100;
   1:  PR[GP1:91,1] = PR[GP1:90,1] + -49.651;
   1:  PR[GP1:91,2] = PR[GP1:90,2] + -14.815;
   1:L PR[91] 10mm/sec CNT100;
   1:  PR[GP1:91,1] = PR[GP1:90,1] + -48.340;
   1:  PR[GP1:91,2] = PR[GP1:90,2] + -17.785;
   1:L PR[91] 10mm/sec CNT100;
   1:  PR[GP1:91,1] = PR[GP1:90,1] + -42.327;
   1:  PR[GP1:91,2] = PR[GP1:90,2] + -27.831;
   1:L PR[91] 10mm/sec CNT100;
   1:  PR[GP1:91,1] = PR[GP1:90,1] + -40.061;
   1:  PR[GP1:91,2] = PR[GP1:90,2] + -30.560;
   1:L PR[91] 10mm/sec CNT100;
   1:  PR[GP1:91,1] = PR[GP1:90,1] + -31.242;
   1:  PR[GP1:91,2] = PR[GP1:90,2] + -37.634;
   1:L PR[91] 10mm/sec CNT100;
   1:  PR[GP1:91,1] = PR[GP1:90,1] + -28.367;
   1:  PR[GP1:91,2] = PR[GP1:90,2] + -39.670;
   1:L PR[91] 10mm/sec CNT100;
   1:  PR[GP1:91,1] = PR[GP1:90,1] + -25.079;
   1:  PR[GP1:91,2] = PR[GP1:90,2] + -40.944;
   1:L PR[91] 10mm/sec CNT100;
   1:  PR[GP1:91,1] = PR[GP1:90,1] + -14.553;
   1:  PR[GP1:91,2] = PR[GP1:90,2] + -44.487;
   1:L PR[91] 10mm/sec CNT100;
   1:  PR[GP1:91,1] = PR[GP1:90,1] + -10.666;
   1:  PR[GP1:91,2] = PR[GP1:90,2] + -44.969;
   1:L PR[91] 10mm/sec CNT100;
   1:  PR[GP1:91,1] = PR[GP1:90,1] + -3.726;
   1:  PR[GP1:91,2] = PR[GP1:90,2] + -44.820;
   1:L PR[91] 10mm/sec CNT100;
   1:  PR[GP1:91,1] = PR[GP1:90,1] + -0.213;
   1:  PR[GP1:91,2] = PR[GP1:90,2] + -44.728;
   1:L PR[91] 10mm/sec CNT100;
   1:  PR[GP1:91,1] = PR[GP1:90,1] + 1.034;
   1:L PR[91] 10mm/sec CNT100;
   1:  PR[GP1:91,1] = PR[GP1:90,1] + 4.546;
   1:  PR[GP1:91,2] = PR[GP1:90,2] + -44.820;
   1:L PR[91] 10mm/sec CNT100;
   1:  PR[GP1:91,1] = PR[GP1:90,1] + 11.487;
   1:  PR[GP1:91,2] = PR[GP1:90,2] + -44.969;
   1:L PR[91] 10mm/sec CNT100;
   1:  PR[GP1:91,1] = PR[GP1:90,1] + 15.374;
   1:  PR[GP1:91,2] = PR[GP1:90,2] + -44.487;
   1:L PR[91] 10mm/sec CNT100;
   1:  PR[GP1:91,1] = PR[GP1:90,1] + 25.900;
   1:  PR[GP1:91,2] = PR[GP1:90,2] + -40.944;
   1:L PR[91] 10mm/sec CNT100;
   1:  PR[GP1:91,1] = PR[GP1:90,1] + 29.172;
   1:  PR[GP1:91,2] = PR[GP1:90,2] + -39.676;
   1:L PR[91] 10mm/sec CNT100;
   1:  PR[GP1:91,1] = PR[GP1:90,1] + 38.291;
   1:  PR[GP1:91,2] = PR[GP1:90,2] + -32.386;
   1:L PR[91] 10mm/sec CNT100;
   1:  PR[GP1:91,1] = PR[GP1:90,1] + 40.895;
   1:  PR[GP1:91,2] = PR[GP1:90,2] + -30.543;
   1:L PR[91] 10mm/sec CNT100;
   1:  PR[GP1:91,1] = PR[GP1:90,1] + 43.148;
   1:  PR[GP1:91,2] = PR[GP1:90,2] + -27.828;
   1:L PR[91] 10mm/sec CNT100;
   1:  PR[GP1:91,1] = PR[GP1:90,1] + 49.161;
   1:  PR[GP1:91,2] = PR[GP1:90,2] + -17.788;
   1:L PR[91] 10mm/sec CNT100;
   1:  PR[GP1:91,1] = PR[GP1:90,1] + 50.477;
   1:  PR[GP1:91,2] = PR[GP1:90,2] + -14.807;
   1:L PR[91] 10mm/sec CNT100;
   1:  PR[GP1:91,1] = PR[GP1:90,1] + 52.613;
   1:  PR[GP1:91,2] = PR[GP1:90,2] + -3.087;
   1:L PR[91] 10mm/sec CNT100;
   1:  PR[GP1:91,1] = PR[GP1:90,1] + 53.041;
   1:  PR[GP1:91,2] = PR[GP1:90,2] + -0.017;
   1:L PR[91] 10mm/sec CNT100;
   1:  PR[GP1:91,1] = PR[GP1:90,1] + 50.927;
   1:  PR[GP1:91,2] = PR[GP1:90,2] + 11.545;
   1:L PR[91] 10mm/sec CNT100;
   1:  PR[GP1:91,1] = PR[GP1:90,1] + 50.472;
   1:  PR[GP1:91,2] = PR[GP1:90,2] + 14.810;
   1:L PR[91] 10mm/sec CNT100;
   1:  PR[GP1:91,1] = PR[GP1:90,1] + 49.161;
   1:  PR[GP1:91,2] = PR[GP1:90,2] + 17.780;
   1:L PR[91] 10mm/sec CNT100;
   1:  PR[GP1:91,1] = PR[GP1:90,1] + 43.148;
   1:  PR[GP1:91,2] = PR[GP1:90,2] + 27.820;
   1:L PR[91] 10mm/sec CNT100;
   1:  PR[GP1:91,1] = PR[GP1:90,1] + 40.882;
   1:  PR[GP1:91,2] = PR[GP1:90,2] + 30.549;
   1:L PR[91] 10mm/sec CNT100;
   1:  PR[GP1:91,1] = PR[GP1:90,1] + 32.062;
   1:  PR[GP1:91,2] = PR[GP1:90,2] + 37.626;
   1:L PR[91] 10mm/sec CNT100;
   1:  PR[GP1:91,1] = PR[GP1:90,1] + 29.187;
   1:  PR[GP1:91,2] = PR[GP1:90,2] + 39.661;
   1:L PR[91] 10mm/sec CNT100;
   1:  PR[GP1:91,1] = PR[GP1:90,1] + 25.898;
   1:  PR[GP1:91,2] = PR[GP1:90,2] + 40.936;
   1:L PR[91] 10mm/sec CNT100;
   1:  PR[GP1:91,1] = PR[GP1:90,1] + 15.372;
   1:  PR[GP1:91,2] = PR[GP1:90,2] + 44.479;
   1:L PR[91] 10mm/sec CNT100;
   1:  PR[GP1:91,1] = PR[GP1:90,1] + 11.484;
   1:  PR[GP1:91,2] = PR[GP1:90,2] + 44.960;
   1:L PR[91] 10mm/sec CNT100;
   1:  PR[GP1:91,1] = PR[GP1:90,1] + 4.567;
   1:  PR[GP1:91,2] = PR[GP1:90,2] + 44.812;
   1:L PR[91] 10mm/sec CNT100;
   1:  PR[GP1:91,1] = PR[GP1:90,1] + 1.033;
   1:  PR[GP1:91,2] = PR[GP1:90,2] + 44.719;
   1:L PR[91] 10mm/sec CNT100;
   1:  PR[GP1:91,1] = PR[GP1:90,1] + -0.162;
   1:  PR[GP1:91,2] = PR[GP1:90,2] + 45.067;
   1:  PR[GP1:91,3] = PR[GP1:90,3] + 111.720;
   1:L PR[91] 10mm/sec CNT100;
   1:  PR[GP1:91,1] = PR[GP1:90,1] + -9.855;
   1:  PR[GP1:91,2] = PR[GP1:90,2] + 45.283;
   1:L PR[91] 10mm/sec CNT100;
   1:  PR[GP1:91,1] = PR[GP1:90,1] + -14.339;
   1:  PR[GP1:91,2] = PR[GP1:90,2] + 44.728;
   1:L PR[91] 10mm/sec CNT100;
   1:  PR[GP1:91,1] = PR[GP1:90,1] + -24.095;
   1:  PR[GP1:91,2] = PR[GP1:90,2] + 41.444;
   1:L PR[91] 10mm/sec CNT100;
   1:  PR[GP1:91,1] = PR[GP1:90,1] + -27.956;
   1:  PR[GP1:91,2] = PR[GP1:90,2] + 39.948;
   1:L PR[91] 10mm/sec CNT100;
   1:  PR[GP1:91,1] = PR[GP1:90,1] + -36.408;
   1:  PR[GP1:91,2] = PR[GP1:90,2] + 33.195;
   1:L PR[91] 10mm/sec CNT100;
   1:  PR[GP1:91,1] = PR[GP1:90,1] + -39.548;
   1:  PR[GP1:91,2] = PR[GP1:90,2] + 30.972;
   1:L PR[91] 10mm/sec CNT100;
   1:  PR[GP1:91,1] = PR[GP1:90,1] + -42.274;
   1:  PR[GP1:91,2] = PR[GP1:90,2] + 27.688;
   1:L PR[91] 10mm/sec CNT100;
   1:  PR[GP1:91,1] = PR[GP1:90,1] + -47.847;
   1:  PR[GP1:91,2] = PR[GP1:90,2] + 18.378;
   1:L PR[91] 10mm/sec CNT100;
   1:  PR[GP1:91,1] = PR[GP1:90,1] + -49.470;
   1:  PR[GP1:91,2] = PR[GP1:90,2] + 14.701;
   1:L PR[91] 10mm/sec CNT100;
   1:  PR[GP1:91,1] = PR[GP1:90,1] + -51.450;
   1:  PR[GP1:91,2] = PR[GP1:90,2] + 3.843;
   1:L PR[91] 10mm/sec CNT100;
   1:  PR[GP1:91,1] = PR[GP1:90,1] + -51.985;
   1:  PR[GP1:91,2] = PR[GP1:90,2] + 0.008;
   1:L PR[91] 10mm/sec CNT100;
   1:  PR[GP1:91,1] = PR[GP1:90,1] + -50.026;
   1:  PR[GP1:91,2] = PR[GP1:90,2] + -10.702;
   1:L PR[91] 10mm/sec CNT100;
   1:  PR[GP1:91,1] = PR[GP1:90,1] + -49.465;
   1:  PR[GP1:91,2] = PR[GP1:90,2] + -14.720;
   1:L PR[91] 10mm/sec CNT100;
   1:  PR[GP1:91,1] = PR[GP1:90,1] + -47.847;
   1:  PR[GP1:91,2] = PR[GP1:90,2] + -18.386;
   1:L PR[91] 10mm/sec CNT100;
   1:  PR[GP1:91,1] = PR[GP1:90,1] + -42.275;
   1:  PR[GP1:91,2] = PR[GP1:90,2] + -27.696;
   1:L PR[91] 10mm/sec CNT100;
   1:  PR[GP1:91,1] = PR[GP1:90,1] + -39.537;
   1:  PR[GP1:91,2] = PR[GP1:90,2] + -30.993;
   1:L PR[91] 10mm/sec CNT100;
   1:  PR[GP1:91,1] = PR[GP1:90,1] + -31.364;
   1:  PR[GP1:91,2] = PR[GP1:90,2] + -37.549;
   1:L PR[91] 10mm/sec CNT100;
   1:  PR[GP1:91,1] = PR[GP1:90,1] + -27.974;
   1:  PR[GP1:91,2] = PR[GP1:90,2] + -39.950;
   1:L PR[91] 10mm/sec CNT100;
   1:  PR[GP1:91,1] = PR[GP1:90,1] + -24.097;
   1:  PR[GP1:91,2] = PR[GP1:90,2] + -41.452;
   1:L PR[91] 10mm/sec CNT100;
   1:  PR[GP1:91,1] = PR[GP1:90,1] + -14.342;
   1:  PR[GP1:91,2] = PR[GP1:90,2] + -44.736;
   1:L PR[91] 10mm/sec CNT100;
   1:  PR[GP1:91,1] = PR[GP1:90,1] + -9.858;
   1:  PR[GP1:91,2] = PR[GP1:90,2] + -45.292;
   1:L PR[91] 10mm/sec CNT100;
   1:  PR[GP1:91,1] = PR[GP1:90,1] + -0.163;
   1:  PR[GP1:91,2] = PR[GP1:90,2] + -45.076;
   1:L PR[91] 10mm/sec CNT100;
   1:  PR[GP1:91,1] = PR[GP1:90,1] + 0.983;
   1:L PR[91] 10mm/sec CNT100;
   1:  PR[GP1:91,1] = PR[GP1:90,1] + 10.679;
   1:  PR[GP1:91,2] = PR[GP1:90,2] + -45.292;
   1:L PR[91] 10mm/sec CNT100;
   1:  PR[GP1:91,1] = PR[GP1:90,1] + 15.163;
   1:  PR[GP1:91,2] = PR[GP1:90,2] + -44.736;
   1:L PR[91] 10mm/sec CNT100;
   1:  PR[GP1:91,1] = PR[GP1:90,1] + 24.918;
   1:  PR[GP1:91,2] = PR[GP1:90,2] + -41.452;
   1:L PR[91] 10mm/sec CNT100;
   1:  PR[GP1:91,1] = PR[GP1:90,1] + 28.779;
   1:  PR[GP1:91,2] = PR[GP1:90,2] + -39.956;
   1:L PR[91] 10mm/sec CNT100;
   1:  PR[GP1:91,1] = PR[GP1:90,1] + 37.230;
   1:  PR[GP1:91,2] = PR[GP1:90,2] + -33.201;
   1:L PR[91] 10mm/sec CNT100;
   1:  PR[GP1:91,1] = PR[GP1:90,1] + 40.371;
   1:  PR[GP1:91,2] = PR[GP1:90,2] + -30.977;
   1:L PR[91] 10mm/sec CNT100;
   1:  PR[GP1:91,1] = PR[GP1:90,1] + 43.096;
   1:  PR[GP1:91,2] = PR[GP1:90,2] + -27.693;
   1:L PR[91] 10mm/sec CNT100;
   1:  PR[GP1:91,1] = PR[GP1:90,1] + 48.668;
   1:  PR[GP1:91,2] = PR[GP1:90,2] + -18.389;
   1:L PR[91] 10mm/sec CNT100;
   1:  PR[GP1:91,1] = PR[GP1:90,1] + 50.291;
   1:  PR[GP1:91,2] = PR[GP1:90,2] + -14.712;
   1:L PR[91] 10mm/sec CNT100;
   1:  PR[GP1:91,1] = PR[GP1:90,1] + 52.271;
   1:  PR[GP1:91,2] = PR[GP1:90,2] + -3.851;
   1:L PR[91] 10mm/sec CNT100;
   1:  PR[GP1:91,1] = PR[GP1:90,1] + 52.805;
   1:  PR[GP1:91,2] = PR[GP1:90,2] + -0.017;
   1:L PR[91] 10mm/sec CNT100;
   1:  PR[GP1:91,1] = PR[GP1:90,1] + 50.846;
   1:  PR[GP1:91,2] = PR[GP1:90,2] + 10.698;
   1:L PR[91] 10mm/sec CNT100;
   1:  PR[GP1:91,1] = PR[GP1:90,1] + 50.286;
   1:  PR[GP1:91,2] = PR[GP1:90,2] + 14.716;
   1:L PR[91] 10mm/sec CNT100;
   1:  PR[GP1:91,1] = PR[GP1:90,1] + 48.668;
   1:  PR[GP1:91,2] = PR[GP1:90,2] + 18.381;
   1:L PR[91] 10mm/sec CNT100;
   1:  PR[GP1:91,1] = PR[GP1:90,1] + 43.096;
   1:  PR[GP1:91,2] = PR[GP1:90,2] + 27.685;
   1:L PR[91] 10mm/sec CNT100;
   1:  PR[GP1:91,1] = PR[GP1:90,1] + 40.358;
   1:  PR[GP1:91,2] = PR[GP1:90,2] + 30.983;
   1:L PR[91] 10mm/sec CNT100;
   1:  PR[GP1:91,1] = PR[GP1:90,1] + 32.184;
   1:  PR[GP1:91,2] = PR[GP1:90,2] + 37.541;
   1:L PR[91] 10mm/sec CNT100;
   1:  PR[GP1:91,1] = PR[GP1:90,1] + 28.794;
   1:  PR[GP1:91,2] = PR[GP1:90,2] + 39.942;
   1:L PR[91] 10mm/sec CNT100;
   1:  PR[GP1:91,1] = PR[GP1:90,1] + 24.916;
   1:  PR[GP1:91,2] = PR[GP1:90,2] + 41.444;
   1:L PR[91] 10mm/sec CNT100;
   1:  PR[GP1:91,1] = PR[GP1:90,1] + 15.161;
   1:  PR[GP1:91,2] = PR[GP1:90,2] + 44.728;
   1:L PR[91] 10mm/sec CNT100;
   1:  PR[GP1:91,1] = PR[GP1:90,1] + 10.676;
   1:  PR[GP1:91,2] = PR[GP1:90,2] + 45.283;
   1:L PR[91] 10mm/sec CNT100;
   1:  PR[GP1:91,1] = PR[GP1:90,1] + 0.983;
   1:  PR[GP1:91,2] = PR[GP1:90,2] + 45.067;
   1:L PR[91] 10mm/sec CNT100;
   1:  PR[GP1:91,1] = PR[GP1:90,1] + -0.113;
   1:  PR[GP1:91,2] = PR[GP1:90,2] + 45.414;
   1:  PR[GP1:91,3] = PR[GP1:90,3] + 113.050;
   1:L PR[91] 10mm/sec CNT100;
   1:  PR[GP1:91,1] = PR[GP1:90,1] + -9.047;
   1:  PR[GP1:91,2] = PR[GP1:90,2] + 45.606;
   1:L PR[91] 10mm/sec CNT100;
   1:  PR[GP1:91,1] = PR[GP1:90,1] + -14.129;
   1:  PR[GP1:91,2] = PR[GP1:90,2] + 44.976;
   1:L PR[91] 10mm/sec CNT100;
   1:  PR[GP1:91,1] = PR[GP1:90,1] + -23.113;
   1:  PR[GP1:91,2] = PR[GP1:90,2] + 41.953;
   1:L PR[91] 10mm/sec CNT100;
   1:  PR[GP1:91,1] = PR[GP1:90,1] + -27.563;
   1:  PR[GP1:91,2] = PR[GP1:90,2] + 40.228;
   1:L PR[91] 10mm/sec CNT100;
   1:  PR[GP1:91,1] = PR[GP1:90,1] + -35.347;
   1:  PR[GP1:91,2] = PR[GP1:90,2] + 34.009;
   1:L PR[91] 10mm/sec CNT100;
   1:  PR[GP1:91,1] = PR[GP1:90,1] + -39.024;
   1:  PR[GP1:91,2] = PR[GP1:90,2] + 31.405;
   1:L PR[91] 10mm/sec CNT100;
   1:  PR[GP1:91,1] = PR[GP1:90,1] + -42.222;
   1:  PR[GP1:91,2] = PR[GP1:90,2] + 27.553;
   1:L PR[91] 10mm/sec CNT100;
   1:  PR[GP1:91,1] = PR[GP1:90,1] + -47.354;
   1:  PR[GP1:91,2] = PR[GP1:90,2] + 18.979;
   1:L PR[91] 10mm/sec CNT100;
   1:  PR[GP1:91,1] = PR[GP1:90,1] + -49.285;
   1:  PR[GP1:91,2] = PR[GP1:90,2] + 14.606;
   1:L PR[91] 10mm/sec CNT100;
   1:  PR[GP1:91,1] = PR[GP1:90,1] + -51.108;
   1:  PR[GP1:91,2] = PR[GP1:90,2] + 4.607;
   1:L PR[91] 10mm/sec CNT100;
   1:  PR[GP1:91,1] = PR[GP1:90,1] + -51.749;
   1:  PR[GP1:91,2] = PR[GP1:90,2] + 0.008;
   1:L PR[91] 10mm/sec CNT100;
   1:  PR[GP1:91,1] = PR[GP1:90,1] + -49.945;
   1:  PR[GP1:91,2] = PR[GP1:90,2] + -9.855;
   1:L PR[91] 10mm/sec CNT100;
   1:  PR[GP1:91,1] = PR[GP1:90,1] + -49.280;
   1:  PR[GP1:91,2] = PR[GP1:90,2] + -14.626;
   1:L PR[91] 10mm/sec CNT100;
   1:  PR[GP1:91,1] = PR[GP1:90,1] + -47.354;
   1:  PR[GP1:91,2] = PR[GP1:90,2] + -18.987;
   1:L PR[91] 10mm/sec CNT100;
   1:  PR[GP1:91,1] = PR[GP1:90,1] + -42.223;
   1:  PR[GP1:91,2] = PR[GP1:90,2] + -27.560;
   1:L PR[91] 10mm/sec CNT100;
   1:  PR[GP1:91,1] = PR[GP1:90,1] + -39.013;
   1:  PR[GP1:91,2] = PR[GP1:90,2] + -31.427;
   1:L PR[91] 10mm/sec CNT100;
   1:  PR[GP1:91,1] = PR[GP1:90,1] + -31.486;
   1:  PR[GP1:91,2] = PR[GP1:90,2] + -37.465;
   1:L PR[91] 10mm/sec CNT100;
   1:  PR[GP1:91,1] = PR[GP1:90,1] + -27.581;
   1:  PR[GP1:91,2] = PR[GP1:90,2] + -40.230;
   1:L PR[91] 10mm/sec CNT100;
   1:  PR[GP1:91,1] = PR[GP1:90,1] + -23.115;
   1:  PR[GP1:91,2] = PR[GP1:90,2] + -41.961;
   1:L PR[91] 10mm/sec CNT100;
   1:  PR[GP1:91,1] = PR[GP1:90,1] + -14.131;
   1:  PR[GP1:91,2] = PR[GP1:90,2] + -44.985;
   1:L PR[91] 10mm/sec CNT100;
   1:  PR[GP1:91,1] = PR[GP1:90,1] + -9.049;
   1:  PR[GP1:91,2] = PR[GP1:90,2] + -45.614;
   1:L PR[91] 10mm/sec CNT100;
   1:  PR[GP1:91,1] = PR[GP1:90,1] + -0.114;
   1:  PR[GP1:91,2] = PR[GP1:90,2] + -45.422;
   1:L PR[91] 10mm/sec CNT100;
   1:  PR[GP1:91,1] = PR[GP1:90,1] + 0.934;
   1:L PR[91] 10mm/sec CNT100;
   1:  PR[GP1:91,1] = PR[GP1:90,1] + 9.870;
   1:  PR[GP1:91,2] = PR[GP1:90,2] + -45.614;
   1:L PR[91] 10mm/sec CNT100;
   1:  PR[GP1:91,1] = PR[GP1:90,1] + 14.952;
   1:  PR[GP1:91,2] = PR[GP1:90,2] + -44.985;
   1:L PR[91] 10mm/sec CNT100;
   1:  PR[GP1:91,1] = PR[GP1:90,1] + 23.936;
   1:  PR[GP1:91,2] = PR[GP1:90,2] + -41.960;
   1:L PR[91] 10mm/sec CNT100;
   1:  PR[GP1:91,1] = PR[GP1:90,1] + 28.386;
   1:  PR[GP1:91,2] = PR[GP1:90,2] + -40.236;
   1:L PR[91] 10mm/sec CNT100;
   1:  PR[GP1:91,1] = PR[GP1:90,1] + 36.169;
   1:  PR[GP1:91,2] = PR[GP1:90,2] + -34.015;
   1:L PR[91] 10mm/sec CNT100;
   1:  PR[GP1:91,1] = PR[GP1:90,1] + 39.846;
   1:  PR[GP1:91,2] = PR[GP1:90,2] + -31.411;
   1:L PR[91] 10mm/sec CNT100;
   1:  PR[GP1:91,1] = PR[GP1:90,1] + 43.044;
   1:  PR[GP1:91,2] = PR[GP1:90,2] + -27.558;
   1:L PR[91] 10mm/sec CNT100;
   1:  PR[GP1:91,1] = PR[GP1:90,1] + 48.175;
   1:  PR[GP1:91,2] = PR[GP1:90,2] + -18.990;
   1:L PR[91] 10mm/sec CNT100;
   1:  PR[GP1:91,1] = PR[GP1:90,1] + 50.106;
   1:  PR[GP1:91,2] = PR[GP1:90,2] + -14.618;
   1:L PR[91] 10mm/sec CNT100;
   1:  PR[GP1:91,1] = PR[GP1:90,1] + 51.928;
   1:  PR[GP1:91,2] = PR[GP1:90,2] + -4.615;
   1:L PR[91] 10mm/sec CNT100;
   1:  PR[GP1:91,1] = PR[GP1:90,1] + 52.570;
   1:  PR[GP1:91,2] = PR[GP1:90,2] + -0.017;
   1:L PR[91] 10mm/sec CNT100;
   1:  PR[GP1:91,1] = PR[GP1:90,1] + 50.766;
   1:  PR[GP1:91,2] = PR[GP1:90,2] + 9.850;
   1:L PR[91] 10mm/sec CNT100;
   1:  PR[GP1:91,1] = PR[GP1:90,1] + 50.100;
   1:  PR[GP1:91,2] = PR[GP1:90,2] + 14.621;
   1:L PR[91] 10mm/sec CNT100;
